KUKA KRL program: repair_test.src, repair_test.dat

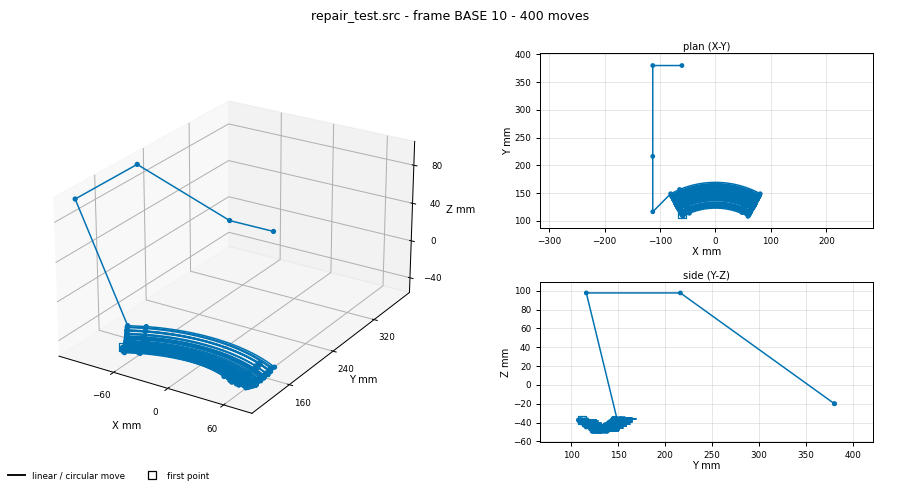
[picture p0: tool path of repair_test.src in frame BASE 10, 400 of 403 moves have a stored position in this frame; points joined in program order, loops and branches not executed]
--- repair_test.src ---
&ACCESS RVP1
&REL 1217
&PARAM WOPTRAJECTORYID = 2
&PARAM WOPTEMPLATENAME = WopCoreTemplatePath
&PARAM DISKPATH = KRC:\R1\Program\Working Paths
DEF  repair_test ( )

;FOLD INI
InitWopCoreSrc(#Init_Trajectory)
;ENDFOLD (INI)

;FOLD Manual mode
IF X_Rob_InManu THEN
;Write here the code executed only in manual mode

ENDIF
;ENDFOLD

X_Prod_En_Cours[2]=TRUE

;FOLD PTP PT_LoopPos1 Vel=10 % DEFAULT Tool[1]:Gun Base[0];%{PE}
;FOLD Parameters ;%{h}
;Params IlfProvider=kukaroboter.basistech.inlineforms.movement.old; Kuka.IsGlobalPoint=False; Kuka.PointName=PT_LoopPos1; Kuka.BlendingEnabled=False; Kuka.MoveDataPtpName=DEFAULT; Kuka.VelocityPtp=10; Kuka.CurrentCDSetIndex=0; Kuka.MovementParameterFieldEnabled=True; IlfCommand=PTP
;ENDFOLD
$BWDSTART = FALSE
PDAT_ACT = PDEFAULT
FDAT_ACT = FPT_LoopPos1
BAS(#PTP_PARAMS, 10.0)
SET_CD_PARAMS (0)
PTP XPT_LoopPos1
;ENDFOLD



;FOLD CHECK DAT-FILE GENERATION NUMBER
  IF APP_GENNUMBER <> 215375 THEN
    LOOP
      MsgQuit("InconsistenceSRCandDAT",,,,1)
      HALT
    ENDLOOP
  ENDIF
;ENDFOLD

;fold Jobinfo
;Job information: repair_test
;Product : 3.1.0.28784
;Date: 2026-09-17-14_00
;Project name: repair_test
;Author: Alhadi Zidan
;Company: CRITT-TJFU
;Division: CSAMProj
;Comment: Autogenerated CSAM Path
;endfold

; --- GLOBAL BLENDING OVERRIDES ---
$APO.CDIS = 1.0  ; Distance blending radius (mm)
$APO.CVEL = 100  ; Velocity blending (%)
$APO.CORI = 5.0  ; Orientation blending (degrees)
$ADVANCE = 5
;FOLD PTP P0 Vel=100 % P0 Tool[2] Base[10] ;%{PE}
;FOLD Parameters ;%{h}
;Params IlfProvider=kukaroboter.basistech.inlineforms.movement.old; Kuka.IsGlobalPoint=False; Kuka.PointName=P0; Kuka.BlendingEnabled=FALSE; Kuka.MoveDataName=PDATP0; Kuka.VelocityPath=100; Kuka.CurrentCDSetIndex=0; Kuka.MovementParameterFieldEnabled=True; IlfCommand=PTP
;ENDFOLD
$BWDSTART = FALSE
PDAT_ACT=PPDATP0
FDAT_ACT=FP0
BAS (#PTP_PARAMS,100)
SET_CD_PARAMS (0)
PTP XP0

;ENDFOLD
Routine_0()
;FOLD PTP PT_LoopPos1 Vel=60 % DEFAULT Tool[1]:Gun Base[0];%{{PE}}
;FOLD Parameters ;%{{h}}
;Params IlfProvider=kukaroboter.basistech.inlineforms.movement.old; Kuka.IsGlobalPoint=False; Kuka.PointName=PT_LoopPos1; Kuka.BlendingEnabled=False; Kuka.MoveDataPtpName=DEFAULT; Kuka.VelocityPtp=10; Kuka.CurrentCDSetIndex=0; Kuka.MovementParameterFieldEnabled=True; IlfCommand=PTP
;ENDFOLD
$BWDSTART = FALSE
PDAT_ACT = PDEFAULT
FDAT_ACT = FPT_LoopPos1
BAS(#PTP_PARAMS, 60.0)
SET_CD_PARAMS (0)
PTP XPT_LoopPos1
;ENDFOLD
END

; --- Routine for substrate 0 ---
DEF Routine_0()
;FOLD LIN P1 CONT Vel=1 m/s CPDATP1 Tool[2] Base[10] ;%{PE}
;FOLD Parameters ;%{h}
;Params IlfProvider=kukaroboter.basistech.inlineforms.movement.old; Kuka.IsGlobalPoint=False; Kuka.PointName=P1; Kuka.BlendingEnabled=TRUE; Kuka.MoveDataName=CPDATP1; Kuka.VelocityPath=1; Kuka.CurrentCDSetIndex=0; Kuka.MovementParameterFieldEnabled=True; IlfCommand=LIN
;ENDFOLD
$BWDSTART = FALSE
LDAT_ACT=LCPDATP1
FDAT_ACT=FP1
BAS (#CP_PARAMS,1)
SET_CD_PARAMS (0)
LIN XP1 C_DIS

;ENDFOLD
;FOLD CIRC CAux2 CDes2 CONT Vel=0.1 m/s CPDATC2 Tool[2] Base[10] ;%{PE}
;FOLD Parameters ;%{h}
;Params IlfProvider=kukaroboter.basistech.inlineforms.movement.old; Kuka.IsGlobalPoint=False; Kuka.PointName=CDes2; Kuka.BlendingEnabled=TRUE; Kuka.MoveDataName=CPDATC2; Kuka.VelocityPath=0.1; Kuka.CurrentCDSetIndex=0; Kuka.MovementParameterFieldEnabled=True; IlfCommand=LIN
;ENDFOLD
$BWDSTART = FALSE
LDAT_ACT=LCPDATC2
FDAT_ACT=FC2
$ORI_TYPE = #VAR
$CIRC_TYPE = #PATH
BAS (#CP_PARAMS,0.1)
SET_CD_PARAMS (0)
CIRC XCAux2, XCDes2 C_DIS

;ENDFOLD
;FOLD LIN P3 CONT Vel=1 m/s CPDATP3 Tool[2] Base[10] ;%{PE}
;FOLD Parameters ;%{h}
;Params IlfProvider=kukaroboter.basistech.inlineforms.movement.old; Kuka.IsGlobalPoint=False; Kuka.PointName=P3; Kuka.BlendingEnabled=TRUE; Kuka.MoveDataName=CPDATP3; Kuka.VelocityPath=1; Kuka.CurrentCDSetIndex=0; Kuka.MovementParameterFieldEnabled=True; IlfCommand=LIN
;ENDFOLD
$BWDSTART = FALSE
LDAT_ACT=LCPDATP3
FDAT_ACT=FP3
BAS (#CP_PARAMS,1)
SET_CD_PARAMS (0)
LIN XP3 C_DIS

;ENDFOLD
;FOLD LIN P4 CONT Vel=1 m/s CPDATP4 Tool[2] Base[10] ;%{PE}
;FOLD Parameters ;%{h}
;Params IlfProvider=kukaroboter.basistech.inlineforms.movement.old; Kuka.IsGlobalPoint=False; Kuka.PointName=P4; Kuka.BlendingEnabled=TRUE; Kuka.MoveDataName=CPDATP4; Kuka.VelocityPath=1; Kuka.CurrentCDSetIndex=0; Kuka.MovementParameterFieldEnabled=True; IlfCommand=LIN
;ENDFOLD
$BWDSTART = FALSE
LDAT_ACT=LCPDATP4
FDAT_ACT=FP4
BAS (#CP_PARAMS,1)
SET_CD_PARAMS (0)
LIN XP4 C_DIS

;ENDFOLD
;FOLD CIRC CAux5 CDes5 CONT Vel=0.1 m/s CPDATC5 Tool[2] Base[10] ;%{PE}
;FOLD Parameters ;%{h}
;Params IlfProvider=kukaroboter.basistech.inlineforms.movement.old; Kuka.IsGlobalPoint=False; Kuka.PointName=CDes5; Kuka.BlendingEnabled=TRUE; Kuka.MoveDataName=CPDATC5; Kuka.VelocityPath=0.1; Kuka.CurrentCDSetIndex=0; Kuka.MovementParameterFieldEnabled=True; IlfCommand=LIN
;ENDFOLD
$BWDSTART = FALSE
LDAT_ACT=LCPDATC5
FDAT_ACT=FC5
$ORI_TYPE = #VAR
$CIRC_TYPE = #PATH
BAS (#CP_PARAMS,0.1)
SET_CD_PARAMS (0)
CIRC XCAux5, XCDes5 C_DIS

;ENDFOLD
;FOLD LIN P6 CONT Vel=1 m/s CPDATP6 Tool[2] Base[10] ;%{PE}
;FOLD Parameters ;%{h}
;Params IlfProvider=kukaroboter.basistech.inlineforms.movement.old; Kuka.IsGlobalPoint=False; Kuka.PointName=P6; Kuka.BlendingEnabled=TRUE; Kuka.MoveDataName=CPDATP6; Kuka.VelocityPath=1; Kuka.CurrentCDSetIndex=0; Kuka.MovementParameterFieldEnabled=True; IlfCommand=LIN
;ENDFOLD
$BWDSTART = FALSE
LDAT_ACT=LCPDATP6
FDAT_ACT=FP6
BAS (#CP_PARAMS,1)
SET_CD_PARAMS (0)
LIN XP6 C_DIS

;ENDFOLD
;FOLD LIN P7 CONT Vel=1 m/s CPDATP7 Tool[2] Base[10] ;%{PE}
;FOLD Parameters ;%{h}
;Params IlfProvider=kukaroboter.basistech.inlineforms.movement.old; Kuka.IsGlobalPoint=False; Kuka.PointName=P7; Kuka.BlendingEnabled=TRUE; Kuka.MoveDataName=CPDATP7; Kuka.VelocityPath=1; Kuka.CurrentCDSetIndex=0; Kuka.MovementParameterFieldEnabled=True; IlfCommand=LIN
;ENDFOLD
$BWDSTART = FALSE
LDAT_ACT=LCPDATP7
FDAT_ACT=FP7
BAS (#CP_PARAMS,1)
SET_CD_PARAMS (0)
LIN XP7 C_DIS

;ENDFOLD
;FOLD CIRC CAux8 CDes8 CONT Vel=0.1 m/s CPDATC8 Tool[2] Base[10] ;%{PE}
;FOLD Parameters ;%{h}
;Params IlfProvider=kukaroboter.basistech.inlineforms.movement.old; Kuka.IsGlobalPoint=False; Kuka.PointName=CDes8; Kuka.BlendingEnabled=TRUE; Kuka.MoveDataName=CPDATC8; Kuka.VelocityPath=0.1; Kuka.CurrentCDSetIndex=0; Kuka.MovementParameterFieldEnabled=True; IlfCommand=LIN
;ENDFOLD
$BWDSTART = FALSE
LDAT_ACT=LCPDATC8
FDAT_ACT=FC8
$ORI_TYPE = #VAR
$CIRC_TYPE = #PATH
BAS (#CP_PARAMS,0.1)
SET_CD_PARAMS (0)
CIRC XCAux8, XCDes8 C_DIS

;ENDFOLD
;FOLD LIN P9 CONT Vel=1 m/s CPDATP9 Tool[2] Base[10] ;%{PE}
;FOLD Parameters ;%{h}
;Params IlfProvider=kukaroboter.basistech.inlineforms.movement.old; Kuka.IsGlobalPoint=False; Kuka.PointName=P9; Kuka.BlendingEnabled=TRUE; Kuka.MoveDataName=CPDATP9; Kuka.VelocityPath=1; Kuka.CurrentCDSetIndex=0; Kuka.MovementParameterFieldEnabled=True; IlfCommand=LIN
;ENDFOLD
$BWDSTART = FALSE
LDAT_ACT=LCPDATP9
FDAT_ACT=FP9
BAS (#CP_PARAMS,1)
SET_CD_PARAMS (0)
LIN XP9 C_DIS

;ENDFOLD
;FOLD LIN P10 CONT Vel=1 m/s CPDATP10 Tool[2] Base[10] ;%{PE}
;FOLD Parameters ;%{h}
;Params IlfProvider=kukaroboter.basistech.inlineforms.movement.old; Kuka.IsGlobalPoint=False; Kuka.PointName=P10; Kuka.BlendingEnabled=TRUE; Kuka.MoveDataName=CPDATP10; Kuka.VelocityPath=1; Kuka.CurrentCDSetIndex=0; Kuka.MovementParameterFieldEnabled=True; IlfCommand=LIN
;ENDFOLD
$BWDSTART = FALSE
LDAT_ACT=LCPDATP10
FDAT_ACT=FP10
BAS (#CP_PARAMS,1)
SET_CD_PARAMS (0)
LIN XP10 C_DIS

;ENDFOLD
;FOLD CIRC CAux11 CDes11 CONT Vel=0.1 m/s CPDATC11 Tool[2] Base[10] ;%{PE}
;FOLD Parameters ;%{h}
;Params IlfProvider=kukaroboter.basistech.inlineforms.movement.old; Kuka.IsGlobalPoint=False; Kuka.PointName=CDes11; Kuka.BlendingEnabled=TRUE; Kuka.MoveDataName=CPDATC11; Kuka.VelocityPath=0.1; Kuka.CurrentCDSetIndex=0; Kuka.MovementParameterFieldEnabled=True; IlfCommand=LIN
;ENDFOLD
$BWDSTART = FALSE
LDAT_ACT=LCPDATC11
FDAT_ACT=FC11
$ORI_TYPE = #VAR
$CIRC_TYPE = #PATH
BAS (#CP_PARAMS,0.1)
SET_CD_PARAMS (0)
CIRC XCAux11, XCDes11 C_DIS

;ENDFOLD
;FOLD LIN P12 CONT Vel=1 m/s CPDATP12 Tool[2] Base[10] ;%{PE}
;FOLD Parameters ;%{h}
;Params IlfProvider=kukaroboter.basistech.inlineforms.movement.old; Kuka.IsGlobalPoint=False; Kuka.PointName=P12; Kuka.BlendingEnabled=TRUE; Kuka.MoveDataName=CPDATP12; Kuka.VelocityPath=1; Kuka.CurrentCDSetIndex=0; Kuka.MovementParameterFieldEnabled=True; IlfCommand=LIN
;ENDFOLD
$BWDSTART = FALSE
LDAT_ACT=LCPDATP12
FDAT_ACT=FP12
BAS (#CP_PARAMS,1)
SET_CD_PARAMS (0)
LIN XP12 C_DIS

;ENDFOLD
;FOLD LIN P13 CONT Vel=1 m/s CPDATP13 Tool[2] Base[10] ;%{PE}
;FOLD Parameters ;%{h}
;Params IlfProvider=kukaroboter.basistech.inlineforms.movement.old; Kuka.IsGlobalPoint=False; Kuka.PointName=P13; Kuka.BlendingEnabled=TRUE; Kuka.MoveDataName=CPDATP13; Kuka.VelocityPath=1; Kuka.CurrentCDSetIndex=0; Kuka.MovementParameterFieldEnabled=True; IlfCommand=LIN
;ENDFOLD
$BWDSTART = FALSE
LDAT_ACT=LCPDATP13
FDAT_ACT=FP13
BAS (#CP_PARAMS,1)
SET_CD_PARAMS (0)
LIN XP13 C_DIS

;ENDFOLD
;FOLD CIRC CAux14 CDes14 CONT Vel=0.1 m/s CPDATC14 Tool[2] Base[10] ;%{PE}
;FOLD Parameters ;%{h}
;Params IlfProvider=kukaroboter.basistech.inlineforms.movement.old; Kuka.IsGlobalPoint=False; Kuka.PointName=CDes14; Kuka.BlendingEnabled=TRUE; Kuka.MoveDataName=CPDATC14; Kuka.VelocityPath=0.1; Kuka.CurrentCDSetIndex=0; Kuka.MovementParameterFieldEnabled=True; IlfCommand=LIN
;ENDFOLD
$BWDSTART = FALSE
LDAT_ACT=LCPDATC14
FDAT_ACT=FC14
$ORI_TYPE = #VAR
$CIRC_TYPE = #PATH
BAS (#CP_PARAMS,0.1)
SET_CD_PARAMS (0)
CIRC XCAux14, XCDes14 C_DIS

;ENDFOLD
;FOLD LIN P15 CONT Vel=1 m/s CPDATP15 Tool[2] Base[10] ;%{PE}
;FOLD Parameters ;%{h}
;Params IlfProvider=kukaroboter.basistech.inlineforms.movement.old; Kuka.IsGlobalPoint=False; Kuka.PointName=P15; Kuka.BlendingEnabled=TRUE; Kuka.MoveDataName=CPDATP15; Kuka.VelocityPath=1; Kuka.CurrentCDSetIndex=0; Kuka.MovementParameterFieldEnabled=True; IlfCommand=LIN
;ENDFOLD
$BWDSTART = FALSE
LDAT_ACT=LCPDATP15
FDAT_ACT=FP15
BAS (#CP_PARAMS,1)
SET_CD_PARAMS (0)
LIN XP15 C_DIS

;ENDFOLD
;FOLD LIN P16 CONT Vel=1 m/s CPDATP16 Tool[2] Base[10] ;%{PE}
;FOLD Parameters ;%{h}
;Params IlfProvider=kukaroboter.basistech.inlineforms.movement.old; Kuka.IsGlobalPoint=False; Kuka.PointName=P16; Kuka.BlendingEnabled=TRUE; Kuka.MoveDataName=CPDATP16; Kuka.VelocityPath=1; Kuka.CurrentCDSetIndex=0; Kuka.MovementParameterFieldEnabled=True; IlfCommand=LIN
;ENDFOLD
$BWDSTART = FALSE
LDAT_ACT=LCPDATP16
FDAT_ACT=FP16
BAS (#CP_PARAMS,1)
SET_CD_PARAMS (0)
LIN XP16 C_DIS

;ENDFOLD
;FOLD CIRC CAux17 CDes17 CONT Vel=0.1 m/s CPDATC17 Tool[2] Base[10] ;%{PE}
;FOLD Parameters ;%{h}
;Params IlfProvider=kukaroboter.basistech.inlineforms.movement.old; Kuka.IsGlobalPoint=False; Kuka.PointName=CDes17; Kuka.BlendingEnabled=TRUE; Kuka.MoveDataName=CPDATC17; Kuka.VelocityPath=0.1; Kuka.CurrentCDSetIndex=0; Kuka.MovementParameterFieldEnabled=True; IlfCommand=LIN
;ENDFOLD
$BWDSTART = FALSE
LDAT_ACT=LCPDATC17
FDAT_ACT=FC17
$ORI_TYPE = #VAR
$CIRC_TYPE = #PATH
BAS (#CP_PARAMS,0.1)
SET_CD_PARAMS (0)
CIRC XCAux17, XCDes17 C_DIS

;ENDFOLD
;FOLD LIN P18 CONT Vel=1 m/s CPDATP18 Tool[2] Base[10] ;%{PE}
;FOLD Parameters ;%{h}
;Params IlfProvider=kukaroboter.basistech.inlineforms.movement.old; Kuka.IsGlobalPoint=False; Kuka.PointName=P18; Kuka.BlendingEnabled=TRUE; Kuka.MoveDataName=CPDATP18; Kuka.VelocityPath=1; Kuka.CurrentCDSetIndex=0; Kuka.MovementParameterFieldEnabled=True; IlfCommand=LIN
;ENDFOLD
$BWDSTART = FALSE
LDAT_ACT=LCPDATP18
FDAT_ACT=FP18
BAS (#CP_PARAMS,1)
SET_CD_PARAMS (0)
LIN XP18 C_DIS

;ENDFOLD
;FOLD LIN P19 CONT Vel=1 m/s CPDATP19 Tool[2] Base[10] ;%{PE}
;FOLD Parameters ;%{h}
;Params IlfProvider=kukaroboter.basistech.inlineforms.movement.old; Kuka.IsGlobalPoint=False; Kuka.PointName=P19; Kuka.BlendingEnabled=TRUE; Kuka.MoveDataName=CPDATP19; Kuka.VelocityPath=1; Kuka.CurrentCDSetIndex=0; Kuka.MovementParameterFieldEnabled=True; IlfCommand=LIN
;ENDFOLD
$BWDSTART = FALSE
LDAT_ACT=LCPDATP19
FDAT_ACT=FP19
BAS (#CP_PARAMS,1)
SET_CD_PARAMS (0)
LIN XP19 C_DIS

;ENDFOLD
;FOLD CIRC CAux20 CDes20 CONT Vel=0.1 m/s CPDATC20 Tool[2] Base[10] ;%{PE}
;FOLD Parameters ;%{h}
;Params IlfProvider=kukaroboter.basistech.inlineforms.movement.old; Kuka.IsGlobalPoint=False; Kuka.PointName=CDes20; Kuka.BlendingEnabled=TRUE; Kuka.MoveDataName=CPDATC20; Kuka.VelocityPath=0.1; Kuka.CurrentCDSetIndex=0; Kuka.MovementParameterFieldEnabled=True; IlfCommand=LIN
;ENDFOLD
$BWDSTART = FALSE
LDAT_ACT=LCPDATC20
FDAT_ACT=FC20
$ORI_TYPE = #VAR
$CIRC_TYPE = #PATH
BAS (#CP_PARAMS,0.1)
SET_CD_PARAMS (0)
CIRC XCAux20, XCDes20 C_DIS

;ENDFOLD
;FOLD LIN P21 CONT Vel=1 m/s CPDATP21 Tool[2] Base[10] ;%{PE}
;FOLD Parameters ;%{h}
;Params IlfProvider=kukaroboter.basistech.inlineforms.movement.old; Kuka.IsGlobalPoint=False; Kuka.PointName=P21; Kuka.BlendingEnabled=TRUE; Kuka.MoveDataName=CPDATP21; Kuka.VelocityPath=1; Kuka.CurrentCDSetIndex=0; Kuka.MovementParameterFieldEnabled=True; IlfCommand=LIN
;ENDFOLD
$BWDSTART = FALSE
LDAT_ACT=LCPDATP21
FDAT_ACT=FP21
BAS (#CP_PARAMS,1)
SET_CD_PARAMS (0)
LIN XP21 C_DIS

;ENDFOLD
;FOLD LIN P22 CONT Vel=1 m/s CPDATP22 Tool[2] Base[10] ;%{PE}
;FOLD Parameters ;%{h}
;Params IlfProvider=kukaroboter.basistech.inlineforms.movement.old; Kuka.IsGlobalPoint=False; Kuka.PointName=P22; Kuka.BlendingEnabled=TRUE; Kuka.MoveDataName=CPDATP22; Kuka.VelocityPath=1; Kuka.CurrentCDSetIndex=0; Kuka.MovementParameterFieldEnabled=True; IlfCommand=LIN
;ENDFOLD
$BWDSTART = FALSE
LDAT_ACT=LCPDATP22
FDAT_ACT=FP22
BAS (#CP_PARAMS,1)
SET_CD_PARAMS (0)
LIN XP22 C_DIS

;ENDFOLD
;FOLD CIRC CAux23 CDes23 CONT Vel=0.1 m/s CPDATC23 Tool[2] Base[10] ;%{PE}
;FOLD Parameters ;%{h}
;Params IlfProvider=kukaroboter.basistech.inlineforms.movement.old; Kuka.IsGlobalPoint=False; Kuka.PointName=CDes23; Kuka.BlendingEnabled=TRUE; Kuka.MoveDataName=CPDATC23; Kuka.VelocityPath=0.1; Kuka.CurrentCDSetIndex=0; Kuka.MovementParameterFieldEnabled=True; IlfCommand=LIN
;ENDFOLD
$BWDSTART = FALSE
LDAT_ACT=LCPDATC23
FDAT_ACT=FC23
$ORI_TYPE = #VAR
$CIRC_TYPE = #PATH
BAS (#CP_PARAMS,0.1)
SET_CD_PARAMS (0)
CIRC XCAux23, XCDes23 C_DIS

;ENDFOLD
;FOLD LIN P24 CONT Vel=1 m/s CPDATP24 Tool[2] Base[10] ;%{PE}
;FOLD Parameters ;%{h}
;Params IlfProvider=kukaroboter.basistech.inlineforms.movement.old; Kuka.IsGlobalPoint=False; Kuka.PointName=P24; Kuka.BlendingEnabled=TRUE; Kuka.MoveDataName=CPDATP24; Kuka.VelocityPath=1; Kuka.CurrentCDSetIndex=0; Kuka.MovementParameterFieldEnabled=True; IlfCommand=LIN
;ENDFOLD
$BWDSTART = FALSE
LDAT_ACT=LCPDATP24
FDAT_ACT=FP24
BAS (#CP_PARAMS,1)
SET_CD_PARAMS (0)
LIN XP24 C_DIS

;ENDFOLD
;FOLD LIN P25 CONT Vel=1 m/s CPDATP25 Tool[2] Base[10] ;%{PE}
;FOLD Parameters ;%{h}
;Params IlfProvider=kukaroboter.basistech.inlineforms.movement.old; Kuka.IsGlobalPoint=False; Kuka.PointName=P25; Kuka.BlendingEnabled=TRUE; Kuka.MoveDataName=CPDATP25; Kuka.VelocityPath=1; Kuka.CurrentCDSetIndex=0; Kuka.MovementParameterFieldEnabled=True; IlfCommand=LIN
;ENDFOLD
$BWDSTART = FALSE
LDAT_ACT=LCPDATP25
FDAT_ACT=FP25
BAS (#CP_PARAMS,1)
SET_CD_PARAMS (0)
LIN XP25 C_DIS

;ENDFOLD
;FOLD CIRC CAux26 CDes26 CONT Vel=0.1 m/s CPDATC26 Tool[2] Base[10] ;%{PE}
;FOLD Parameters ;%{h}
;Params IlfProvider=kukaroboter.basistech.inlineforms.movement.old; Kuka.IsGlobalPoint=False; Kuka.PointName=CDes26; Kuka.BlendingEnabled=TRUE; Kuka.MoveDataName=CPDATC26; Kuka.VelocityPath=0.1; Kuka.CurrentCDSetIndex=0; Kuka.MovementParameterFieldEnabled=True; IlfCommand=LIN
;ENDFOLD
$BWDSTART = FALSE
LDAT_ACT=LCPDATC26
FDAT_ACT=FC26
$ORI_TYPE = #VAR
$CIRC_TYPE = #PATH
BAS (#CP_PARAMS,0.1)
SET_CD_PARAMS (0)
CIRC XCAux26, XCDes26 C_DIS

;ENDFOLD
;FOLD LIN P27 CONT Vel=1 m/s CPDATP27 Tool[2] Base[10] ;%{PE}
;FOLD Parameters ;%{h}
;Params IlfProvider=kukaroboter.basistech.inlineforms.movement.old; Kuka.IsGlobalPoint=False; Kuka.PointName=P27; Kuka.BlendingEnabled=TRUE; Kuka.MoveDataName=CPDATP27; Kuka.VelocityPath=1; Kuka.CurrentCDSetIndex=0; Kuka.MovementParameterFieldEnabled=True; IlfCommand=LIN
;ENDFOLD
$BWDSTART = FALSE
LDAT_ACT=LCPDATP27
FDAT_ACT=FP27
BAS (#CP_PARAMS,1)
SET_CD_PARAMS (0)
LIN XP27 C_DIS

;ENDFOLD
;FOLD LIN P28 CONT Vel=1 m/s CPDATP28 Tool[2] Base[10] ;%{PE}
;FOLD Parameters ;%{h}
;Params IlfProvider=kukaroboter.basistech.inlineforms.movement.old; Kuka.IsGlobalPoint=False; Kuka.PointName=P28; Kuka.BlendingEnabled=TRUE; Kuka.MoveDataName=CPDATP28; Kuka.VelocityPath=1; Kuka.CurrentCDSetIndex=0; Kuka.MovementParameterFieldEnabled=True; IlfCommand=LIN
;ENDFOLD
$BWDSTART = FALSE
LDAT_ACT=LCPDATP28
FDAT_ACT=FP28
BAS (#CP_PARAMS,1)
SET_CD_PARAMS (0)
LIN XP28 C_DIS

;ENDFOLD
;FOLD CIRC CAux29 CDes29 CONT Vel=0.1 m/s CPDATC29 Tool[2] Base[10] ;%{PE}
;FOLD Parameters ;%{h}
;Params IlfProvider=kukaroboter.basistech.inlineforms.movement.old; Kuka.IsGlobalPoint=False; Kuka.PointName=CDes29; Kuka.BlendingEnabled=TRUE; Kuka.MoveDataName=CPDATC29; Kuka.VelocityPath=0.1; Kuka.CurrentCDSetIndex=0; Kuka.MovementParameterFieldEnabled=True; IlfCommand=LIN
;ENDFOLD
$BWDSTART = FALSE
LDAT_ACT=LCPDATC29
FDAT_ACT=FC29
$ORI_TYPE = #VAR
$CIRC_TYPE = #PATH
BAS (#CP_PARAMS,0.1)
SET_CD_PARAMS (0)
CIRC XCAux29, XCDes29 C_DIS

;ENDFOLD
;FOLD LIN P30 CONT Vel=1 m/s CPDATP30 Tool[2] Base[10] ;%{PE}
;FOLD Parameters ;%{h}
;Params IlfProvider=kukaroboter.basistech.inlineforms.movement.old; Kuka.IsGlobalPoint=False; Kuka.PointName=P30; Kuka.BlendingEnabled=TRUE; Kuka.MoveDataName=CPDATP30; Kuka.VelocityPath=1; Kuka.CurrentCDSetIndex=0; Kuka.MovementParameterFieldEnabled=True; IlfCommand=LIN
;ENDFOLD
$BWDSTART = FALSE
LDAT_ACT=LCPDATP30
FDAT_ACT=FP30
BAS (#CP_PARAMS,1)
SET_CD_PARAMS (0)
LIN XP30 C_DIS

;ENDFOLD
;FOLD LIN P31 CONT Vel=1 m/s CPDATP31 Tool[2] Base[10] ;%{PE}
;FOLD Parameters ;%{h}
;Params IlfProvider=kukaroboter.basistech.inlineforms.movement.old; Kuka.IsGlobalPoint=False; Kuka.PointName=P31; Kuka.BlendingEnabled=TRUE; Kuka.MoveDataName=CPDATP31; Kuka.VelocityPath=1; Kuka.CurrentCDSetIndex=0; Kuka.MovementParameterFieldEnabled=True; IlfCommand=LIN
;ENDFOLD
$BWDSTART = FALSE
LDAT_ACT=LCPDATP31
FDAT_ACT=FP31
BAS (#CP_PARAMS,1)
SET_CD_PARAMS (0)
LIN XP31 C_DIS

;ENDFOLD
;FOLD CIRC CAux32 CDes32 CONT Vel=0.1 m/s CPDATC32 Tool[2] Base[10] ;%{PE}
;FOLD Parameters ;%{h}
;Params IlfProvider=kukaroboter.basistech.inlineforms.movement.old; Kuka.IsGlobalPoint=False; Kuka.PointName=CDes32; Kuka.BlendingEnabled=TRUE; Kuka.MoveDataName=CPDATC32; Kuka.VelocityPath=0.1; Kuka.CurrentCDSetIndex=0; Kuka.MovementParameterFieldEnabled=True; IlfCommand=LIN
;ENDFOLD
$BWDSTART = FALSE
LDAT_ACT=LCPDATC32
FDAT_ACT=FC32
$ORI_TYPE = #VAR
$CIRC_TYPE = #PATH
BAS (#CP_PARAMS,0.1)
SET_CD_PARAMS (0)
CIRC XCAux32, XCDes32 C_DIS

;ENDFOLD
;FOLD LIN P33 CONT Vel=1 m/s CPDATP33 Tool[2] Base[10] ;%{PE}
;FOLD Parameters ;%{h}
;Params IlfProvider=kukaroboter.basistech.inlineforms.movement.old; Kuka.IsGlobalPoint=False; Kuka.PointName=P33; Kuka.BlendingEnabled=TRUE; Kuka.MoveDataName=CPDATP33; Kuka.VelocityPath=1; Kuka.CurrentCDSetIndex=0; Kuka.MovementParameterFieldEnabled=True; IlfCommand=LIN
;ENDFOLD
$BWDSTART = FALSE
LDAT_ACT=LCPDATP33
FDAT_ACT=FP33
BAS (#CP_PARAMS,1)
SET_CD_PARAMS (0)
LIN XP33 C_DIS

;ENDFOLD
;FOLD LIN P34 CONT Vel=1 m/s CPDATP34 Tool[2] Base[10] ;%{PE}
;FOLD Parameters ;%{h}
;Params IlfProvider=kukaroboter.basistech.inlineforms.movement.old; Kuka.IsGlobalPoint=False; Kuka.PointName=P34; Kuka.BlendingEnabled=TRUE; Kuka.MoveDataName=CPDATP34; Kuka.VelocityPath=1; Kuka.CurrentCDSetIndex=0; Kuka.MovementParameterFieldEnabled=True; IlfCommand=LIN
;ENDFOLD
$BWDSTART = FALSE
LDAT_ACT=LCPDATP34
FDAT_ACT=FP34
BAS (#CP_PARAMS,1)
SET_CD_PARAMS (0)
LIN XP34 C_DIS

;ENDFOLD
;FOLD CIRC CAux35 CDes35 CONT Vel=0.1 m/s CPDATC35 Tool[2] Base[10] ;%{PE}
;FOLD Parameters ;%{h}
;Params IlfProvider=kukaroboter.basistech.inlineforms.movement.old; Kuka.IsGlobalPoint=False; Kuka.PointName=CDes35; Kuka.BlendingEnabled=TRUE; Kuka.MoveDataName=CPDATC35; Kuka.VelocityPath=0.1; Kuka.CurrentCDSetIndex=0; Kuka.MovementParameterFieldEnabled=True; IlfCommand=LIN
;ENDFOLD
$BWDSTART = FALSE
LDAT_ACT=LCPDATC35
FDAT_ACT=FC35
$ORI_TYPE = #VAR
$CIRC_TYPE = #PATH
BAS (#CP_PARAMS,0.1)
SET_CD_PARAMS (0)
CIRC XCAux35, XCDes35 C_DIS

;ENDFOLD
;FOLD LIN P36 CONT Vel=1 m/s CPDATP36 Tool[2] Base[10] ;%{PE}
;FOLD Parameters ;%{h}
;Params IlfProvider=kukaroboter.basistech.inlineforms.movement.old; Kuka.IsGlobalPoint=False; Kuka.PointName=P36; Kuka.BlendingEnabled=TRUE; Kuka.MoveDataName=CPDATP36; Kuka.VelocityPath=1; Kuka.CurrentCDSetIndex=0; Kuka.MovementParameterFieldEnabled=True; IlfCommand=LIN
;ENDFOLD
$BWDSTART = FALSE
LDAT_ACT=LCPDATP36
FDAT_ACT=FP36
BAS (#CP_PARAMS,1)
SET_CD_PARAMS (0)
LIN XP36 C_DIS

;ENDFOLD
;FOLD LIN P37 CONT Vel=1 m/s CPDATP37 Tool[2] Base[10] ;%{PE}
;FOLD Parameters ;%{h}
;Params IlfProvider=kukaroboter.basistech.inlineforms.movement.old; Kuka.IsGlobalPoint=False; Kuka.PointName=P37; Kuka.BlendingEnabled=TRUE; Kuka.MoveDataName=CPDATP37; Kuka.VelocityPath=1; Kuka.CurrentCDSetIndex=0; Kuka.MovementParameterFieldEnabled=True; IlfCommand=LIN
;ENDFOLD
$BWDSTART = FALSE
LDAT_ACT=LCPDATP37
FDAT_ACT=FP37
BAS (#CP_PARAMS,1)
SET_CD_PARAMS (0)
LIN XP37 C_DIS

;ENDFOLD
;FOLD CIRC CAux38 CDes38 CONT Vel=0.1 m/s CPDATC38 Tool[2] Base[10] ;%{PE}
;FOLD Parameters ;%{h}
;Params IlfProvider=kukaroboter.basistech.inlineforms.movement.old; Kuka.IsGlobalPoint=False; Kuka.PointName=CDes38; Kuka.BlendingEnabled=TRUE; Kuka.MoveDataName=CPDATC38; Kuka.VelocityPath=0.1; Kuka.CurrentCDSetIndex=0; Kuka.MovementParameterFieldEnabled=True; IlfCommand=LIN
;ENDFOLD
$BWDSTART = FALSE
LDAT_ACT=LCPDATC38
FDAT_ACT=FC38
$ORI_TYPE = #VAR
$CIRC_TYPE = #PATH
BAS (#CP_PARAMS,0.1)
SET_CD_PARAMS (0)
CIRC XCAux38, XCDes38 C_DIS

;ENDFOLD
;FOLD LIN P39 CONT Vel=1 m/s CPDATP39 Tool[2] Base[10] ;%{PE}
;FOLD Parameters ;%{h}
;Params IlfProvider=kukaroboter.basistech.inlineforms.movement.old; Kuka.IsGlobalPoint=False; Kuka.PointName=P39; Kuka.BlendingEnabled=TRUE; Kuka.MoveDataName=CPDATP39; Kuka.VelocityPath=1; Kuka.CurrentCDSetIndex=0; Kuka.MovementParameterFieldEnabled=True; IlfCommand=LIN
;ENDFOLD
$BWDSTART = FALSE
LDAT_ACT=LCPDATP39
FDAT_ACT=FP39
BAS (#CP_PARAMS,1)
SET_CD_PARAMS (0)
LIN XP39 C_DIS

;ENDFOLD
;FOLD LIN P40 CONT Vel=1 m/s CPDATP40 Tool[2] Base[10] ;%{PE}
;FOLD Parameters ;%{h}
;Params IlfProvider=kukaroboter.basistech.inlineforms.movement.old; Kuka.IsGlobalPoint=False; Kuka.PointName=P40; Kuka.BlendingEnabled=TRUE; Kuka.MoveDataName=CPDATP40; Kuka.VelocityPath=1; Kuka.CurrentCDSetIndex=0; Kuka.MovementParameterFieldEnabled=True; IlfCommand=LIN
;ENDFOLD
$BWDSTART = FALSE
LDAT_ACT=LCPDATP40
FDAT_ACT=FP40
BAS (#CP_PARAMS,1)
SET_CD_PARAMS (0)
LIN XP40 C_DIS

;ENDFOLD
;FOLD CIRC CAux41 CDes41 CONT Vel=0.1 m/s CPDATC41 Tool[2] Base[10] ;%{PE}
;FOLD Parameters ;%{h}
;Params IlfProvider=kukaroboter.basistech.inlineforms.movement.old; Kuka.IsGlobalPoint=False; Kuka.PointName=CDes41; Kuka.BlendingEnabled=TRUE; Kuka.MoveDataName=CPDATC41; Kuka.VelocityPath=0.1; Kuka.CurrentCDSetIndex=0; Kuka.MovementParameterFieldEnabled=True; IlfCommand=LIN
;ENDFOLD
$BWDSTART = FALSE
LDAT_ACT=LCPDATC41
FDAT_ACT=FC41
$ORI_TYPE = #VAR
$CIRC_TYPE = #PATH
BAS (#CP_PARAMS,0.1)
SET_CD_PARAMS (0)
CIRC XCAux41, XCDes41 C_DIS

;ENDFOLD
;FOLD LIN P42 CONT Vel=1 m/s CPDATP42 Tool[2] Base[10] ;%{PE}
;FOLD Parameters ;%{h}
;Params IlfProvider=kukaroboter.basistech.inlineforms.movement.old; Kuka.IsGlobalPoint=False; Kuka.PointName=P42; Kuka.BlendingEnabled=TRUE; Kuka.MoveDataName=CPDATP42; Kuka.VelocityPath=1; Kuka.CurrentCDSetIndex=0; Kuka.MovementParameterFieldEnabled=True; IlfCommand=LIN
;ENDFOLD
$BWDSTART = FALSE
LDAT_ACT=LCPDATP42
FDAT_ACT=FP42
BAS (#CP_PARAMS,1)
SET_CD_PARAMS (0)
LIN XP42 C_DIS

;ENDFOLD
;FOLD LIN P43 CONT Vel=1 m/s CPDATP43 Tool[2] Base[10] ;%{PE}
;FOLD Parameters ;%{h}
;Params IlfProvider=kukaroboter.basistech.inlineforms.movement.old; Kuka.IsGlobalPoint=False; Kuka.PointName=P43; Kuka.BlendingEnabled=TRUE; Kuka.MoveDataName=CPDATP43; Kuka.VelocityPath=1; Kuka.CurrentCDSetIndex=0; Kuka.MovementParameterFieldEnabled=True; IlfCommand=LIN
;ENDFOLD
$BWDSTART = FALSE
LDAT_ACT=LCPDATP43
FDAT_ACT=FP43
BAS (#CP_PARAMS,1)
SET_CD_PARAMS (0)
LIN XP43 C_DIS

;ENDFOLD
;FOLD CIRC CAux44 CDes44 CONT Vel=0.1 m/s CPDATC44 Tool[2] Base[10] ;%{PE}
;FOLD Parameters ;%{h}
;Params IlfProvider=kukaroboter.basistech.inlineforms.movement.old; Kuka.IsGlobalPoint=False; Kuka.PointName=CDes44; Kuka.BlendingEnabled=TRUE; Kuka.MoveDataName=CPDATC44; Kuka.VelocityPath=0.1; Kuka.CurrentCDSetIndex=0; Kuka.MovementParameterFieldEnabled=True; IlfCommand=LIN
;ENDFOLD
$BWDSTART = FALSE
LDAT_ACT=LCPDATC44
FDAT_ACT=FC44
$ORI_TYPE = #VAR
$CIRC_TYPE = #PATH
BAS (#CP_PARAMS,0.1)
SET_CD_PARAMS (0)
CIRC XCAux44, XCDes44 C_DIS

;ENDFOLD
;FOLD LIN P45 CONT Vel=1 m/s CPDATP45 Tool[2] Base[10] ;%{PE}
;FOLD Parameters ;%{h}
;Params IlfProvider=kukaroboter.basistech.inlineforms.movement.old; Kuka.IsGlobalPoint=False; Kuka.PointName=P45; Kuka.BlendingEnabled=TRUE; Kuka.MoveDataName=CPDATP45; Kuka.VelocityPath=1; Kuka.CurrentCDSetIndex=0; Kuka.MovementParameterFieldEnabled=True; IlfCommand=LIN
;ENDFOLD
$BWDSTART = FALSE
LDAT_ACT=LCPDATP45
FDAT_ACT=FP45
BAS (#CP_PARAMS,1)
SET_CD_PARAMS (0)
LIN XP45 C_DIS

;ENDFOLD
;FOLD LIN P46 CONT Vel=1 m/s CPDATP46 Tool[2] Base[10] ;%{PE}
;FOLD Parameters ;%{h}
;Params IlfProvider=kukaroboter.basistech.inlineforms.movement.old; Kuka.IsGlobalPoint=False; Kuka.PointName=P46; Kuka.BlendingEnabled=TRUE; Kuka.MoveDataName=CPDATP46; Kuka.VelocityPath=1; Kuka.CurrentCDSetIndex=0; Kuka.MovementParameterFieldEnabled=True; IlfCommand=LIN
;ENDFOLD
$BWDSTART = FALSE
LDAT_ACT=LCPDATP46
FDAT_ACT=FP46
BAS (#CP_PARAMS,1)
SET_CD_PARAMS (0)
LIN XP46 C_DIS

;ENDFOLD
;FOLD CIRC CAux47 CDes47 CONT Vel=0.1 m/s CPDATC47 Tool[2] Base[10] ;%{PE}
;FOLD Parameters ;%{h}
;Params IlfProvider=kukaroboter.basistech.inlineforms.movement.old; Kuka.IsGlobalPoint=False; Kuka.PointName=CDes47; Kuka.BlendingEnabled=TRUE; Kuka.MoveDataName=CPDATC47; Kuka.VelocityPath=0.1; Kuka.CurrentCDSetIndex=0; Kuka.MovementParameterFieldEnabled=True; IlfCommand=LIN
;ENDFOLD
$BWDSTART = FALSE
LDAT_ACT=LCPDATC47
FDAT_ACT=FC47
$ORI_TYPE = #VAR
$CIRC_TYPE = #PATH
BAS (#CP_PARAMS,0.1)
SET_CD_PARAMS (0)
CIRC XCAux47, XCDes47 C_DIS

;ENDFOLD
;FOLD LIN P48 CONT Vel=1 m/s CPDATP48 Tool[2] Base[10] ;%{PE}
;FOLD Parameters ;%{h}
;Params IlfProvider=kukaroboter.basistech.inlineforms.movement.old; Kuka.IsGlobalPoint=False; Kuka.PointName=P48; Kuka.BlendingEnabled=TRUE; Kuka.MoveDataName=CPDATP48; Kuka.VelocityPath=1; Kuka.CurrentCDSetIndex=0; Kuka.MovementParameterFieldEnabled=True; IlfCommand=LIN
;ENDFOLD
$BWDSTART = FALSE
LDAT_ACT=LCPDATP48
FDAT_ACT=FP48
BAS (#CP_PARAMS,1)
SET_CD_PARAMS (0)
LIN XP48 C_DIS

;ENDFOLD
;FOLD LIN P49 CONT Vel=1 m/s CPDATP49 Tool[2] Base[10] ;%{PE}
;FOLD Parameters ;%{h}
;Params IlfProvider=kukaroboter.basistech.inlineforms.movement.old; Kuka.IsGlobalPoint=False; Kuka.PointName=P49; Kuka.BlendingEnabled=TRUE; Kuka.MoveDataName=CPDATP49; Kuka.VelocityPath=1; Kuka.CurrentCDSetIndex=0; Kuka.MovementParameterFieldEnabled=True; IlfCommand=LIN
;ENDFOLD
$BWDSTART = FALSE
LDAT_ACT=LCPDATP49
FDAT_ACT=FP49
BAS (#CP_PARAMS,1)
SET_CD_PARAMS (0)
LIN XP49 C_DIS

;ENDFOLD
;FOLD CIRC CAux50 CDes50 CONT Vel=0.1 m/s CPDATC50 Tool[2] Base[10] ;%{PE}
;FOLD Parameters ;%{h}
;Params IlfProvider=kukaroboter.basistech.inlineforms.movement.old; Kuka.IsGlobalPoint=False; Kuka.PointName=CDes50; Kuka.BlendingEnabled=TRUE; Kuka.MoveDataName=CPDATC50; Kuka.VelocityPath=0.1; Kuka.CurrentCDSetIndex=0; Kuka.MovementParameterFieldEnabled=True; IlfCommand=LIN
;ENDFOLD
$BWDSTART = FALSE
LDAT_ACT=LCPDATC50
FDAT_ACT=FC50
$ORI_TYPE = #VAR
$CIRC_TYPE = #PATH
BAS (#CP_PARAMS,0.1)
SET_CD_PARAMS (0)
CIRC XCAux50, XCDes50 C_DIS

;ENDFOLD
;FOLD LIN P51 CONT Vel=1 m/s CPDATP51 Tool[2] Base[10] ;%{PE}
;FOLD Parameters ;%{h}
;Params IlfProvider=kukaroboter.basistech.inlineforms.movement.old; Kuka.IsGlobalPoint=False; Kuka.PointName=P51; Kuka.BlendingEnabled=TRUE; Kuka.MoveDataName=CPDATP51; Kuka.VelocityPath=1; Kuka.CurrentCDSetIndex=0; Kuka.MovementParameterFieldEnabled=True; IlfCommand=LIN
;ENDFOLD
$BWDSTART = FALSE
LDAT_ACT=LCPDATP51
FDAT_ACT=FP51
BAS (#CP_PARAMS,1)
SET_CD_PARAMS (0)
LIN XP51 C_DIS

;ENDFOLD
;FOLD LIN P52 CONT Vel=1 m/s CPDATP52 Tool[2] Base[10] ;%{PE}
;FOLD Parameters ;%{h}
;Params IlfProvider=kukaroboter.basistech.inlineforms.movement.old; Kuka.IsGlobalPoint=False; Kuka.PointName=P52; Kuka.BlendingEnabled=TRUE; Kuka.MoveDataName=CPDATP52; Kuka.VelocityPath=1; Kuka.CurrentCDSetIndex=0; Kuka.MovementParameterFieldEnabled=True; IlfCommand=LIN
;ENDFOLD
$BWDSTART = FALSE
LDAT_ACT=LCPDATP52
FDAT_ACT=FP52
BAS (#CP_PARAMS,1)
SET_CD_PARAMS (0)
LIN XP52 C_DIS

;ENDFOLD
;FOLD CIRC CAux53 CDes53 CONT Vel=0.1 m/s CPDATC53 Tool[2] Base[10] ;%{PE}
;FOLD Parameters ;%{h}
;Params IlfProvider=kukaroboter.basistech.inlineforms.movement.old; Kuka.IsGlobalPoint=False; Kuka.PointName=CDes53; Kuka.BlendingEnabled=TRUE; Kuka.MoveDataName=CPDATC53; Kuka.VelocityPath=0.1; Kuka.CurrentCDSetIndex=0; Kuka.MovementParameterFieldEnabled=True; IlfCommand=LIN
;ENDFOLD
$BWDSTART = FALSE
LDAT_ACT=LCPDATC53
FDAT_ACT=FC53
$ORI_TYPE = #VAR
$CIRC_TYPE = #PATH
BAS (#CP_PARAMS,0.1)
SET_CD_PARAMS (0)
CIRC XCAux53, XCDes53 C_DIS

;ENDFOLD
;FOLD LIN P54 CONT Vel=1 m/s CPDATP54 Tool[2] Base[10] ;%{PE}
;FOLD Parameters ;%{h}
;Params IlfProvider=kukaroboter.basistech.inlineforms.movement.old; Kuka.IsGlobalPoint=False; Kuka.PointName=P54; Kuka.BlendingEnabled=TRUE; Kuka.MoveDataName=CPDATP54; Kuka.VelocityPath=1; Kuka.CurrentCDSetIndex=0; Kuka.MovementParameterFieldEnabled=True; IlfCommand=LIN
;ENDFOLD
$BWDSTART = FALSE
LDAT_ACT=LCPDATP54
FDAT_ACT=FP54
BAS (#CP_PARAMS,1)
SET_CD_PARAMS (0)
LIN XP54 C_DIS

;ENDFOLD
;FOLD LIN P55 CONT Vel=1 m/s CPDATP55 Tool[2] Base[10] ;%{PE}
;FOLD Parameters ;%{h}
;Params IlfProvider=kukaroboter.basistech.inlineforms.movement.old; Kuka.IsGlobalPoint=False; Kuka.PointName=P55; Kuka.BlendingEnabled=TRUE; Kuka.MoveDataName=CPDATP55; Kuka.VelocityPath=1; Kuka.CurrentCDSetIndex=0; Kuka.MovementParameterFieldEnabled=True; IlfCommand=LIN
;ENDFOLD
$BWDSTART = FALSE
LDAT_ACT=LCPDATP55
FDAT_ACT=FP55
BAS (#CP_PARAMS,1)
SET_CD_PARAMS (0)
LIN XP55 C_DIS

;ENDFOLD
;FOLD CIRC CAux56 CDes56 CONT Vel=0.1 m/s CPDATC56 Tool[2] Base[10] ;%{PE}
;FOLD Parameters ;%{h}
;Params IlfProvider=kukaroboter.basistech.inlineforms.movement.old; Kuka.IsGlobalPoint=False; Kuka.PointName=CDes56; Kuka.BlendingEnabled=TRUE; Kuka.MoveDataName=CPDATC56; Kuka.VelocityPath=0.1; Kuka.CurrentCDSetIndex=0; Kuka.MovementParameterFieldEnabled=True; IlfCommand=LIN
;ENDFOLD
$BWDSTART = FALSE
LDAT_ACT=LCPDATC56
FDAT_ACT=FC56
$ORI_TYPE = #VAR
$CIRC_TYPE = #PATH
BAS (#CP_PARAMS,0.1)
SET_CD_PARAMS (0)
CIRC XCAux56, XCDes56 C_DIS

;ENDFOLD
;FOLD LIN P57 CONT Vel=1 m/s CPDATP57 Tool[2] Base[10] ;%{PE}
;FOLD Parameters ;%{h}
;Params IlfProvider=kukaroboter.basistech.inlineforms.movement.old; Kuka.IsGlobalPoint=False; Kuka.PointName=P57; Kuka.BlendingEnabled=TRUE; Kuka.MoveDataName=CPDATP57; Kuka.VelocityPath=1; Kuka.CurrentCDSetIndex=0; Kuka.MovementParameterFieldEnabled=True; IlfCommand=LIN
;ENDFOLD
$BWDSTART = FALSE
LDAT_ACT=LCPDATP57
FDAT_ACT=FP57
BAS (#CP_PARAMS,1)
SET_CD_PARAMS (0)
LIN XP57 C_DIS

;ENDFOLD
;FOLD LIN P58 CONT Vel=1 m/s CPDATP58 Tool[2] Base[10] ;%{PE}
;FOLD Parameters ;%{h}
;Params IlfProvider=kukaroboter.basistech.inlineforms.movement.old; Kuka.IsGlobalPoint=False; Kuka.PointName=P58; Kuka.BlendingEnabled=TRUE; Kuka.MoveDataName=CPDATP58; Kuka.VelocityPath=1; Kuka.CurrentCDSetIndex=0; Kuka.MovementParameterFieldEnabled=True; IlfCommand=LIN
;ENDFOLD
$BWDSTART = FALSE
LDAT_ACT=LCPDATP58
FDAT_ACT=FP58
BAS (#CP_PARAMS,1)
SET_CD_PARAMS (0)
LIN XP58 C_DIS

;ENDFOLD
;FOLD CIRC CAux59 CDes59 CONT Vel=0.1 m/s CPDATC59 Tool[2] Base[10] ;%{PE}
;FOLD Parameters ;%{h}
;Params IlfProvider=kukaroboter.basistech.inlineforms.movement.old; Kuka.IsGlobalPoint=False; Kuka.PointName=CDes59; Kuka.BlendingEnabled=TRUE; Kuka.MoveDataName=CPDATC59; Kuka.VelocityPath=0.1; Kuka.CurrentCDSetIndex=0; Kuka.MovementParameterFieldEnabled=True; IlfCommand=LIN
;ENDFOLD
$BWDSTART = FALSE
LDAT_ACT=LCPDATC59
FDAT_ACT=FC59
$ORI_TYPE = #VAR
$CIRC_TYPE = #PATH
BAS (#CP_PARAMS,0.1)
SET_CD_PARAMS (0)
CIRC XCAux59, XCDes59 C_DIS

;ENDFOLD
;FOLD LIN P60 CONT Vel=1 m/s CPDATP60 Tool[2] Base[10] ;%{PE}
;FOLD Parameters ;%{h}
;Params IlfProvider=kukaroboter.basistech.inlineforms.movement.old; Kuka.IsGlobalPoint=False; Kuka.PointName=P60; Kuka.BlendingEnabled=TRUE; Kuka.MoveDataName=CPDATP60; Kuka.VelocityPath=1; Kuka.CurrentCDSetIndex=0; Kuka.MovementParameterFieldEnabled=True; IlfCommand=LIN
;ENDFOLD
$BWDSTART = FALSE
LDAT_ACT=LCPDATP60
FDAT_ACT=FP60
BAS (#CP_PARAMS,1)
SET_CD_PARAMS (0)
LIN XP60 C_DIS

;ENDFOLD
;FOLD LIN P61 CONT Vel=1 m/s CPDATP61 Tool[2] Base[10] ;%{PE}
;FOLD Parameters ;%{h}
;Params IlfProvider=kukaroboter.basistech.inlineforms.movement.old; Kuka.IsGlobalPoint=False; Kuka.PointName=P61; Kuka.BlendingEnabled=TRUE; Kuka.MoveDataName=CPDATP61; Kuka.VelocityPath=1; Kuka.CurrentCDSetIndex=0; Kuka.MovementParameterFieldEnabled=True; IlfCommand=LIN
;ENDFOLD
$BWDSTART = FALSE
LDAT_ACT=LCPDATP61
FDAT_ACT=FP61
BAS (#CP_PARAMS,1)
SET_CD_PARAMS (0)
LIN XP61 C_DIS

;ENDFOLD
;FOLD CIRC CAux62 CDes62 CONT Vel=0.1 m/s CPDATC62 Tool[2] Base[10] ;%{PE}
;FOLD Parameters ;%{h}
;Params IlfProvider=kukaroboter.basistech.inlineforms.movement.old; Kuka.IsGlobalPoint=False; Kuka.PointName=CDes62; Kuka.BlendingEnabled=TRUE; Kuka.MoveDataName=CPDATC62; Kuka.VelocityPath=0.1; Kuka.CurrentCDSetIndex=0; Kuka.MovementParameterFieldEnabled=True; IlfCommand=LIN
;ENDFOLD
$BWDSTART = FALSE
LDAT_ACT=LCPDATC62
FDAT_ACT=FC62
$ORI_TYPE = #VAR
$CIRC_TYPE = #PATH
BAS (#CP_PARAMS,0.1)
SET_CD_PARAMS (0)
CIRC XCAux62, XCDes62 C_DIS

;ENDFOLD
;FOLD LIN P63 CONT Vel=1 m/s CPDATP63 Tool[2] Base[10] ;%{PE}
;FOLD Parameters ;%{h}
;Params IlfProvider=kukaroboter.basistech.inlineforms.movement.old; Kuka.IsGlobalPoint=False; Kuka.PointName=P63; Kuka.BlendingEnabled=TRUE; Kuka.MoveDataName=CPDATP63; Kuka.VelocityPath=1; Kuka.CurrentCDSetIndex=0; Kuka.MovementParameterFieldEnabled=True; IlfCommand=LIN
;ENDFOLD
$BWDSTART = FALSE
LDAT_ACT=LCPDATP63
FDAT_ACT=FP63
BAS (#CP_PARAMS,1)
SET_CD_PARAMS (0)
LIN XP63 C_DIS

;ENDFOLD
;FOLD LIN P64 CONT Vel=1 m/s CPDATP64 Tool[2] Base[10] ;%{PE}
;FOLD Parameters ;%{h}
;Params IlfProvider=kukaroboter.basistech.inlineforms.movement.old; Kuka.IsGlobalPoint=False; Kuka.PointName=P64; Kuka.BlendingEnabled=TRUE; Kuka.MoveDataName=CPDATP64; Kuka.VelocityPath=1; Kuka.CurrentCDSetIndex=0; Kuka.MovementParameterFieldEnabled=True; IlfCommand=LIN
;ENDFOLD
$BWDSTART = FALSE
LDAT_ACT=LCPDATP64
FDAT_ACT=FP64
BAS (#CP_PARAMS,1)
SET_CD_PARAMS (0)
LIN XP64 C_DIS

;ENDFOLD
;FOLD CIRC CAux65 CDes65 CONT Vel=0.1 m/s CPDATC65 Tool[2] Base[10] ;%{PE}
;FOLD Parameters ;%{h}
;Params IlfProvider=kukaroboter.basistech.inlineforms.movement.old; Kuka.IsGlobalPoint=False; Kuka.PointName=CDes65; Kuka.BlendingEnabled=TRUE; Kuka.MoveDataName=CPDATC65; Kuka.VelocityPath=0.1; Kuka.CurrentCDSetIndex=0; Kuka.MovementParameterFieldEnabled=True; IlfCommand=LIN
;ENDFOLD
$BWDSTART = FALSE
LDAT_ACT=LCPDATC65
FDAT_ACT=FC65
$ORI_TYPE = #VAR
$CIRC_TYPE = #PATH
BAS (#CP_PARAMS,0.1)
SET_CD_PARAMS (0)
CIRC XCAux65, XCDes65 C_DIS

;ENDFOLD
;FOLD LIN P66 CONT Vel=1 m/s CPDATP66 Tool[2] Base[10] ;%{PE}
;FOLD Parameters ;%{h}
;Params IlfProvider=kukaroboter.basistech.inlineforms.movement.old; Kuka.IsGlobalPoint=False; Kuka.PointName=P66; Kuka.BlendingEnabled=TRUE; Kuka.MoveDataName=CPDATP66; Kuka.VelocityPath=1; Kuka.CurrentCDSetIndex=0; Kuka.MovementParameterFieldEnabled=True; IlfCommand=LIN
;ENDFOLD
$BWDSTART = FALSE
LDAT_ACT=LCPDATP66
FDAT_ACT=FP66
BAS (#CP_PARAMS,1)
SET_CD_PARAMS (0)
LIN XP66 C_DIS

;ENDFOLD
;FOLD LIN P67 CONT Vel=1 m/s CPDATP67 Tool[2] Base[10] ;%{PE}
;FOLD Parameters ;%{h}
;Params IlfProvider=kukaroboter.basistech.inlineforms.movement.old; Kuka.IsGlobalPoint=False; Kuka.PointName=P67; Kuka.BlendingEnabled=TRUE; Kuka.MoveDataName=CPDATP67; Kuka.VelocityPath=1; Kuka.CurrentCDSetIndex=0; Kuka.MovementParameterFieldEnabled=True; IlfCommand=LIN
;ENDFOLD
$BWDSTART = FALSE
LDAT_ACT=LCPDATP67
FDAT_ACT=FP67
BAS (#CP_PARAMS,1)
SET_CD_PARAMS (0)
LIN XP67 C_DIS

;ENDFOLD
;FOLD CIRC CAux68 CDes68 CONT Vel=0.1 m/s CPDATC68 Tool[2] Base[10] ;%{PE}
;FOLD Parameters ;%{h}
;Params IlfProvider=kukaroboter.basistech.inlineforms.movement.old; Kuka.IsGlobalPoint=False; Kuka.PointName=CDes68; Kuka.BlendingEnabled=TRUE; Kuka.MoveDataName=CPDATC68; Kuka.VelocityPath=0.1; Kuka.CurrentCDSetIndex=0; Kuka.MovementParameterFieldEnabled=True; IlfCommand=LIN
;ENDFOLD
$BWDSTART = FALSE
LDAT_ACT=LCPDATC68
FDAT_ACT=FC68
$ORI_TYPE = #VAR
$CIRC_TYPE = #PATH
BAS (#CP_PARAMS,0.1)
SET_CD_PARAMS (0)
CIRC XCAux68, XCDes68 C_DIS

;ENDFOLD
;FOLD LIN P69 CONT Vel=1 m/s CPDATP69 Tool[2] Base[10] ;%{PE}
;FOLD Parameters ;%{h}
;Params IlfProvider=kukaroboter.basistech.inlineforms.movement.old; Kuka.IsGlobalPoint=False; Kuka.PointName=P69; Kuka.BlendingEnabled=TRUE; Kuka.MoveDataName=CPDATP69; Kuka.VelocityPath=1; Kuka.CurrentCDSetIndex=0; Kuka.MovementParameterFieldEnabled=True; IlfCommand=LIN
;ENDFOLD
$BWDSTART = FALSE
LDAT_ACT=LCPDATP69
FDAT_ACT=FP69
BAS (#CP_PARAMS,1)
SET_CD_PARAMS (0)
LIN XP69 C_DIS

;ENDFOLD
;FOLD LIN P70 CONT Vel=1 m/s CPDATP70 Tool[2] Base[10] ;%{PE}
;FOLD Parameters ;%{h}
;Params IlfProvider=kukaroboter.basistech.inlineforms.movement.old; Kuka.IsGlobalPoint=False; Kuka.PointName=P70; Kuka.BlendingEnabled=TRUE; Kuka.MoveDataName=CPDATP70; Kuka.VelocityPath=1; Kuka.CurrentCDSetIndex=0; Kuka.MovementParameterFieldEnabled=True; IlfCommand=LIN
;ENDFOLD
$BWDSTART = FALSE
LDAT_ACT=LCPDATP70
FDAT_ACT=FP70
BAS (#CP_PARAMS,1)
SET_CD_PARAMS (0)
LIN XP70 C_DIS

;ENDFOLD
;FOLD CIRC CAux71 CDes71 CONT Vel=0.1 m/s CPDATC71 Tool[2] Base[10] ;%{PE}
;FOLD Parameters ;%{h}
;Params IlfProvider=kukaroboter.basistech.inlineforms.movement.old; Kuka.IsGlobalPoint=False; Kuka.PointName=CDes71; Kuka.BlendingEnabled=TRUE; Kuka.MoveDataName=CPDATC71; Kuka.VelocityPath=0.1; Kuka.CurrentCDSetIndex=0; Kuka.MovementParameterFieldEnabled=True; IlfCommand=LIN
;ENDFOLD
$BWDSTART = FALSE
LDAT_ACT=LCPDATC71
FDAT_ACT=FC71
$ORI_TYPE = #VAR
$CIRC_TYPE = #PATH
BAS (#CP_PARAMS,0.1)
SET_CD_PARAMS (0)
CIRC XCAux71, XCDes71 C_DIS

;ENDFOLD
;FOLD LIN P72 CONT Vel=1 m/s CPDATP72 Tool[2] Base[10] ;%{PE}
;FOLD Parameters ;%{h}
;Params IlfProvider=kukaroboter.basistech.inlineforms.movement.old; Kuka.IsGlobalPoint=False; Kuka.PointName=P72; Kuka.BlendingEnabled=TRUE; Kuka.MoveDataName=CPDATP72; Kuka.VelocityPath=1; Kuka.CurrentCDSetIndex=0; Kuka.MovementParameterFieldEnabled=True; IlfCommand=LIN
;ENDFOLD
$BWDSTART = FALSE
LDAT_ACT=LCPDATP72
FDAT_ACT=FP72
BAS (#CP_PARAMS,1)
SET_CD_PARAMS (0)
LIN XP72 C_DIS

;ENDFOLD
;FOLD LIN P73 CONT Vel=1 m/s CPDATP73 Tool[2] Base[10] ;%{PE}
;FOLD Parameters ;%{h}
;Params IlfProvider=kukaroboter.basistech.inlineforms.movement.old; Kuka.IsGlobalPoint=False; Kuka.PointName=P73; Kuka.BlendingEnabled=TRUE; Kuka.MoveDataName=CPDATP73; Kuka.VelocityPath=1; Kuka.CurrentCDSetIndex=0; Kuka.MovementParameterFieldEnabled=True; IlfCommand=LIN
;ENDFOLD
$BWDSTART = FALSE
LDAT_ACT=LCPDATP73
FDAT_ACT=FP73
BAS (#CP_PARAMS,1)
SET_CD_PARAMS (0)
LIN XP73 C_DIS

;ENDFOLD
;FOLD CIRC CAux74 CDes74 CONT Vel=0.1 m/s CPDATC74 Tool[2] Base[10] ;%{PE}
;FOLD Parameters ;%{h}
;Params IlfProvider=kukaroboter.basistech.inlineforms.movement.old; Kuka.IsGlobalPoint=False; Kuka.PointName=CDes74; Kuka.BlendingEnabled=TRUE; Kuka.MoveDataName=CPDATC74; Kuka.VelocityPath=0.1; Kuka.CurrentCDSetIndex=0; Kuka.MovementParameterFieldEnabled=True; IlfCommand=LIN
;ENDFOLD
$BWDSTART = FALSE
LDAT_ACT=LCPDATC74
FDAT_ACT=FC74
$ORI_TYPE = #VAR
$CIRC_TYPE = #PATH
BAS (#CP_PARAMS,0.1)
SET_CD_PARAMS (0)
CIRC XCAux74, XCDes74 C_DIS

;ENDFOLD
;FOLD LIN P75 CONT Vel=1 m/s CPDATP75 Tool[2] Base[10] ;%{PE}
;FOLD Parameters ;%{h}
;Params IlfProvider=kukaroboter.basistech.inlineforms.movement.old; Kuka.IsGlobalPoint=False; Kuka.PointName=P75; Kuka.BlendingEnabled=TRUE; Kuka.MoveDataName=CPDATP75; Kuka.VelocityPath=1; Kuka.CurrentCDSetIndex=0; Kuka.MovementParameterFieldEnabled=True; IlfCommand=LIN
;ENDFOLD
$BWDSTART = FALSE
LDAT_ACT=LCPDATP75
FDAT_ACT=FP75
BAS (#CP_PARAMS,1)
SET_CD_PARAMS (0)
LIN XP75 C_DIS

;ENDFOLD
;FOLD LIN P76 CONT Vel=1 m/s CPDATP76 Tool[2] Base[10] ;%{PE}
;FOLD Parameters ;%{h}
;Params IlfProvider=kukaroboter.basistech.inlineforms.movement.old; Kuka.IsGlobalPoint=False; Kuka.PointName=P76; Kuka.BlendingEnabled=TRUE; Kuka.MoveDataName=CPDATP76; Kuka.VelocityPath=1; Kuka.CurrentCDSetIndex=0; Kuka.MovementParameterFieldEnabled=True; IlfCommand=LIN
;ENDFOLD
$BWDSTART = FALSE
LDAT_ACT=LCPDATP76
FDAT_ACT=FP76
BAS (#CP_PARAMS,1)
SET_CD_PARAMS (0)
LIN XP76 C_DIS

;ENDFOLD
;FOLD CIRC CAux77 CDes77 CONT Vel=0.1 m/s CPDATC77 Tool[2] Base[10] ;%{PE}
;FOLD Parameters ;%{h}
;Params IlfProvider=kukaroboter.basistech.inlineforms.movement.old; Kuka.IsGlobalPoint=False; Kuka.PointName=CDes77; Kuka.BlendingEnabled=TRUE; Kuka.MoveDataName=CPDATC77; Kuka.VelocityPath=0.1; Kuka.CurrentCDSetIndex=0; Kuka.MovementParameterFieldEnabled=True; IlfCommand=LIN
;ENDFOLD
$BWDSTART = FALSE
LDAT_ACT=LCPDATC77
FDAT_ACT=FC77
$ORI_TYPE = #VAR
$CIRC_TYPE = #PATH
BAS (#CP_PARAMS,0.1)
SET_CD_PARAMS (0)
CIRC XCAux77, XCDes77 C_DIS

;ENDFOLD
;FOLD LIN P78 CONT Vel=1 m/s CPDATP78 Tool[2] Base[10] ;%{PE}
;FOLD Parameters ;%{h}
;Params IlfProvider=kukaroboter.basistech.inlineforms.movement.old; Kuka.IsGlobalPoint=False; Kuka.PointName=P78; Kuka.BlendingEnabled=TRUE; Kuka.MoveDataName=CPDATP78; Kuka.VelocityPath=1; Kuka.CurrentCDSetIndex=0; Kuka.MovementParameterFieldEnabled=True; IlfCommand=LIN
;ENDFOLD
$BWDSTART = FALSE
LDAT_ACT=LCPDATP78
FDAT_ACT=FP78
BAS (#CP_PARAMS,1)
SET_CD_PARAMS (0)
LIN XP78 C_DIS

;ENDFOLD
;FOLD LIN P79 CONT Vel=1 m/s CPDATP79 Tool[2] Base[10] ;%{PE}
;FOLD Parameters ;%{h}
;Params IlfProvider=kukaroboter.basistech.inlineforms.movement.old; Kuka.IsGlobalPoint=False; Kuka.PointName=P79; Kuka.BlendingEnabled=TRUE; Kuka.MoveDataName=CPDATP79; Kuka.VelocityPath=1; Kuka.CurrentCDSetIndex=0; Kuka.MovementParameterFieldEnabled=True; IlfCommand=LIN
;ENDFOLD
$BWDSTART = FALSE
LDAT_ACT=LCPDATP79
FDAT_ACT=FP79
BAS (#CP_PARAMS,1)
SET_CD_PARAMS (0)
LIN XP79 C_DIS

;ENDFOLD
;FOLD CIRC CAux80 CDes80 CONT Vel=0.1 m/s CPDATC80 Tool[2] Base[10] ;%{PE}
;FOLD Parameters ;%{h}
;Params IlfProvider=kukaroboter.basistech.inlineforms.movement.old; Kuka.IsGlobalPoint=False; Kuka.PointName=CDes80; Kuka.BlendingEnabled=TRUE; Kuka.MoveDataName=CPDATC80; Kuka.VelocityPath=0.1; Kuka.CurrentCDSetIndex=0; Kuka.MovementParameterFieldEnabled=True; IlfCommand=LIN
;ENDFOLD
$BWDSTART = FALSE
LDAT_ACT=LCPDATC80
FDAT_ACT=FC80
$ORI_TYPE = #VAR
$CIRC_TYPE = #PATH
BAS (#CP_PARAMS,0.1)
SET_CD_PARAMS (0)
CIRC XCAux80, XCDes80 C_DIS

;ENDFOLD
;FOLD LIN P81 CONT Vel=1 m/s CPDATP81 Tool[2] Base[10] ;%{PE}
;FOLD Parameters ;%{h}
;Params IlfProvider=kukaroboter.basistech.inlineforms.movement.old; Kuka.IsGlobalPoint=False; Kuka.PointName=P81; Kuka.BlendingEnabled=TRUE; Kuka.MoveDataName=CPDATP81; Kuka.VelocityPath=1; Kuka.CurrentCDSetIndex=0; Kuka.MovementParameterFieldEnabled=True; IlfCommand=LIN
;ENDFOLD
$BWDSTART = FALSE
LDAT_ACT=LCPDATP81
FDAT_ACT=FP81
BAS (#CP_PARAMS,1)
SET_CD_PARAMS (0)
LIN XP81 C_DIS

;ENDFOLD
;FOLD LIN P82 CONT Vel=1 m/s CPDATP82 Tool[2] Base[10] ;%{PE}
;FOLD Parameters ;%{h}
;Params IlfProvider=kukaroboter.basistech.inlineforms.movement.old; Kuka.IsGlobalPoint=False; Kuka.PointName=P82; Kuka.BlendingEnabled=TRUE; Kuka.MoveDataName=CPDATP82; Kuka.VelocityPath=1; Kuka.CurrentCDSetIndex=0; Kuka.MovementParameterFieldEnabled=True; IlfCommand=LIN
;ENDFOLD
$BWDSTART = FALSE
LDAT_ACT=LCPDATP82
FDAT_ACT=FP82
BAS (#CP_PARAMS,1)
SET_CD_PARAMS (0)
LIN XP82 C_DIS

;ENDFOLD
;FOLD CIRC CAux83 CDes83 CONT Vel=0.1 m/s CPDATC83 Tool[2] Base[10] ;%{PE}
;FOLD Parameters ;%{h}
;Params IlfProvider=kukaroboter.basistech.inlineforms.movement.old; Kuka.IsGlobalPoint=False; Kuka.PointName=CDes83; Kuka.BlendingEnabled=TRUE; Kuka.MoveDataName=CPDATC83; Kuka.VelocityPath=0.1; Kuka.CurrentCDSetIndex=0; Kuka.MovementParameterFieldEnabled=True; IlfCommand=LIN
;ENDFOLD
$BWDSTART = FALSE
LDAT_ACT=LCPDATC83
FDAT_ACT=FC83
$ORI_TYPE = #VAR
$CIRC_TYPE = #PATH
BAS (#CP_PARAMS,0.1)
SET_CD_PARAMS (0)
CIRC XCAux83, XCDes83 C_DIS

;ENDFOLD
;FOLD LIN P84 CONT Vel=1 m/s CPDATP84 Tool[2] Base[10] ;%{PE}
;FOLD Parameters ;%{h}
;Params IlfProvider=kukaroboter.basistech.inlineforms.movement.old; Kuka.IsGlobalPoint=False; Kuka.PointName=P84; Kuka.BlendingEnabled=TRUE; Kuka.MoveDataName=CPDATP84; Kuka.VelocityPath=1; Kuka.CurrentCDSetIndex=0; Kuka.MovementParameterFieldEnabled=True; IlfCommand=LIN
;ENDFOLD
$BWDSTART = FALSE
LDAT_ACT=LCPDATP84
FDAT_ACT=FP84
BAS (#CP_PARAMS,1)
SET_CD_PARAMS (0)
LIN XP84 C_DIS

;ENDFOLD
;FOLD LIN P85 CONT Vel=1 m/s CPDATP85 Tool[2] Base[10] ;%{PE}
;FOLD Parameters ;%{h}
;Params IlfProvider=kukaroboter.basistech.inlineforms.movement.old; Kuka.IsGlobalPoint=False; Kuka.PointName=P85; Kuka.BlendingEnabled=TRUE; Kuka.MoveDataName=CPDATP85; Kuka.VelocityPath=1; Kuka.CurrentCDSetIndex=0; Kuka.MovementParameterFieldEnabled=True; IlfCommand=LIN
;ENDFOLD
$BWDSTART = FALSE
LDAT_ACT=LCPDATP85
FDAT_ACT=FP85
BAS (#CP_PARAMS,1)
SET_CD_PARAMS (0)
LIN XP85 C_DIS

;ENDFOLD
;FOLD CIRC CAux86 CDes86 CONT Vel=0.1 m/s CPDATC86 Tool[2] Base[10] ;%{PE}
;FOLD Parameters ;%{h}
;Params IlfProvider=kukaroboter.basistech.inlineforms.movement.old; Kuka.IsGlobalPoint=False; Kuka.PointName=CDes86; Kuka.BlendingEnabled=TRUE; Kuka.MoveDataName=CPDATC86; Kuka.VelocityPath=0.1; Kuka.CurrentCDSetIndex=0; Kuka.MovementParameterFieldEnabled=True; IlfCommand=LIN
;ENDFOLD
$BWDSTART = FALSE
LDAT_ACT=LCPDATC86
FDAT_ACT=FC86
$ORI_TYPE = #VAR
$CIRC_TYPE = #PATH
BAS (#CP_PARAMS,0.1)
SET_CD_PARAMS (0)
CIRC XCAux86, XCDes86 C_DIS

;ENDFOLD
;FOLD LIN P87 CONT Vel=1 m/s CPDATP87 Tool[2] Base[10] ;%{PE}
;FOLD Parameters ;%{h}
;Params IlfProvider=kukaroboter.basistech.inlineforms.movement.old; Kuka.IsGlobalPoint=False; Kuka.PointName=P87; Kuka.BlendingEnabled=TRUE; Kuka.MoveDataName=CPDATP87; Kuka.VelocityPath=1; Kuka.CurrentCDSetIndex=0; Kuka.MovementParameterFieldEnabled=True; IlfCommand=LIN
;ENDFOLD
$BWDSTART = FALSE
LDAT_ACT=LCPDATP87
FDAT_ACT=FP87
BAS (#CP_PARAMS,1)
SET_CD_PARAMS (0)
LIN XP87 C_DIS

;ENDFOLD
;FOLD LIN P88 CONT Vel=1 m/s CPDATP88 Tool[2] Base[10] ;%{PE}
;FOLD Parameters ;%{h}
;Params IlfProvider=kukaroboter.basistech.inlineforms.movement.old; Kuka.IsGlobalPoint=False; Kuka.PointName=P88; Kuka.BlendingEnabled=TRUE; Kuka.MoveDataName=CPDATP88; Kuka.VelocityPath=1; Kuka.CurrentCDSetIndex=0; Kuka.MovementParameterFieldEnabled=True; IlfCommand=LIN
;ENDFOLD
$BWDSTART = FALSE
LDAT_ACT=LCPDATP88
FDAT_ACT=FP88
BAS (#CP_PARAMS,1)
SET_CD_PARAMS (0)
LIN XP88 C_DIS

;ENDFOLD
;FOLD CIRC CAux89 CDes89 CONT Vel=0.1 m/s CPDATC89 Tool[2] Base[10] ;%{PE}
;FOLD Parameters ;%{h}
;Params IlfProvider=kukaroboter.basistech.inlineforms.movement.old; Kuka.IsGlobalPoint=False; Kuka.PointName=CDes89; Kuka.BlendingEnabled=TRUE; Kuka.MoveDataName=CPDATC89; Kuka.VelocityPath=0.1; Kuka.CurrentCDSetIndex=0; Kuka.MovementParameterFieldEnabled=True; IlfCommand=LIN
;ENDFOLD
$BWDSTART = FALSE
LDAT_ACT=LCPDATC89
FDAT_ACT=FC89
$ORI_TYPE = #VAR
$CIRC_TYPE = #PATH
BAS (#CP_PARAMS,0.1)
SET_CD_PARAMS (0)
CIRC XCAux89, XCDes89 C_DIS

;ENDFOLD
;FOLD LIN P90 CONT Vel=1 m/s CPDATP90 Tool[2] Base[10] ;%{PE}
;FOLD Parameters ;%{h}
;Params IlfProvider=kukaroboter.basistech.inlineforms.movement.old; Kuka.IsGlobalPoint=False; Kuka.PointName=P90; Kuka.BlendingEnabled=TRUE; Kuka.MoveDataName=CPDATP90; Kuka.VelocityPath=1; Kuka.CurrentCDSetIndex=0; Kuka.MovementParameterFieldEnabled=True; IlfCommand=LIN
;ENDFOLD
$BWDSTART = FALSE
LDAT_ACT=LCPDATP90
FDAT_ACT=FP90
BAS (#CP_PARAMS,1)
SET_CD_PARAMS (0)
LIN XP90 C_DIS

;ENDFOLD
;FOLD LIN P91 CONT Vel=1 m/s CPDATP91 Tool[2] Base[10] ;%{PE}
;FOLD Parameters ;%{h}
;Params IlfProvider=kukaroboter.basistech.inlineforms.movement.old; Kuka.IsGlobalPoint=False; Kuka.PointName=P91; Kuka.BlendingEnabled=TRUE; Kuka.MoveDataName=CPDATP91; Kuka.VelocityPath=1; Kuka.CurrentCDSetIndex=0; Kuka.MovementParameterFieldEnabled=True; IlfCommand=LIN
;ENDFOLD
$BWDSTART = FALSE
LDAT_ACT=LCPDATP91
FDAT_ACT=FP91
BAS (#CP_PARAMS,1)
SET_CD_PARAMS (0)
LIN XP91 C_DIS

;ENDFOLD
;FOLD CIRC CAux92 CDes92 CONT Vel=0.1 m/s CPDATC92 Tool[2] Base[10] ;%{PE}
;FOLD Parameters ;%{h}
;Params IlfProvider=kukaroboter.basistech.inlineforms.movement.old; Kuka.IsGlobalPoint=False; Kuka.PointName=CDes92; Kuka.BlendingEnabled=TRUE; Kuka.MoveDataName=CPDATC92; Kuka.VelocityPath=0.1; Kuka.CurrentCDSetIndex=0; Kuka.MovementParameterFieldEnabled=True; IlfCommand=LIN
;ENDFOLD
$BWDSTART = FALSE
LDAT_ACT=LCPDATC92
FDAT_ACT=FC92
$ORI_TYPE = #VAR
$CIRC_TYPE = #PATH
BAS (#CP_PARAMS,0.1)
SET_CD_PARAMS (0)
CIRC XCAux92, XCDes92 C_DIS

;ENDFOLD
;FOLD LIN P93 CONT Vel=1 m/s CPDATP93 Tool[2] Base[10] ;%{PE}
;FOLD Parameters ;%{h}
;Params IlfProvider=kukaroboter.basistech.inlineforms.movement.old; Kuka.IsGlobalPoint=False; Kuka.PointName=P93; Kuka.BlendingEnabled=TRUE; Kuka.MoveDataName=CPDATP93; Kuka.VelocityPath=1; Kuka.CurrentCDSetIndex=0; Kuka.MovementParameterFieldEnabled=True; IlfCommand=LIN
;ENDFOLD
$BWDSTART = FALSE
LDAT_ACT=LCPDATP93
FDAT_ACT=FP93
BAS (#CP_PARAMS,1)
SET_CD_PARAMS (0)
LIN XP93 C_DIS

;ENDFOLD
;FOLD LIN P94 CONT Vel=1 m/s CPDATP94 Tool[2] Base[10] ;%{PE}
;FOLD Parameters ;%{h}
;Params IlfProvider=kukaroboter.basistech.inlineforms.movement.old; Kuka.IsGlobalPoint=False; Kuka.PointName=P94; Kuka.BlendingEnabled=TRUE; Kuka.MoveDataName=CPDATP94; Kuka.VelocityPath=1; Kuka.CurrentCDSetIndex=0; Kuka.MovementParameterFieldEnabled=True; IlfCommand=LIN
;ENDFOLD
$BWDSTART = FALSE
LDAT_ACT=LCPDATP94
FDAT_ACT=FP94
BAS (#CP_PARAMS,1)
SET_CD_PARAMS (0)
LIN XP94 C_DIS

;ENDFOLD
;FOLD CIRC CAux95 CDes95 CONT Vel=0.1 m/s CPDATC95 Tool[2] Base[10] ;%{PE}
;FOLD Parameters ;%{h}
;Params IlfProvider=kukaroboter.basistech.inlineforms.movement.old; Kuka.IsGlobalPoint=False; Kuka.PointName=CDes95; Kuka.BlendingEnabled=TRUE; Kuka.MoveDataName=CPDATC95; Kuka.VelocityPath=0.1; Kuka.CurrentCDSetIndex=0; Kuka.MovementParameterFieldEnabled=True; IlfCommand=LIN
;ENDFOLD
$BWDSTART = FALSE
LDAT_ACT=LCPDATC95
FDAT_ACT=FC95
$ORI_TYPE = #VAR
$CIRC_TYPE = #PATH
BAS (#CP_PARAMS,0.1)
SET_CD_PARAMS (0)
CIRC XCAux95, XCDes95 C_DIS

;ENDFOLD
;FOLD LIN P96 CONT Vel=1 m/s CPDATP96 Tool[2] Base[10] ;%{PE}
;FOLD Parameters ;%{h}
;Params IlfProvider=kukaroboter.basistech.inlineforms.movement.old; Kuka.IsGlobalPoint=False; Kuka.PointName=P96; Kuka.BlendingEnabled=TRUE; Kuka.MoveDataName=CPDATP96; Kuka.VelocityPath=1; Kuka.CurrentCDSetIndex=0; Kuka.MovementParameterFieldEnabled=True; IlfCommand=LIN
;ENDFOLD
$BWDSTART = FALSE
LDAT_ACT=LCPDATP96
FDAT_ACT=FP96
BAS (#CP_PARAMS,1)
SET_CD_PARAMS (0)
LIN XP96 C_DIS

;ENDFOLD
;FOLD LIN P97 CONT Vel=1 m/s CPDATP97 Tool[2] Base[10] ;%{PE}
;FOLD Parameters ;%{h}
;Params IlfProvider=kukaroboter.basistech.inlineforms.movement.old; Kuka.IsGlobalPoint=False; Kuka.PointName=P97; Kuka.BlendingEnabled=TRUE; Kuka.MoveDataName=CPDATP97; Kuka.VelocityPath=1; Kuka.CurrentCDSetIndex=0; Kuka.MovementParameterFieldEnabled=True; IlfCommand=LIN
;ENDFOLD
$BWDSTART = FALSE
LDAT_ACT=LCPDATP97
FDAT_ACT=FP97
BAS (#CP_PARAMS,1)
SET_CD_PARAMS (0)
LIN XP97 C_DIS

;ENDFOLD
;FOLD CIRC CAux98 CDes98 CONT Vel=0.1 m/s CPDATC98 Tool[2] Base[10] ;%{PE}
;FOLD Parameters ;%{h}
;Params IlfProvider=kukaroboter.basistech.inlineforms.movement.old; Kuka.IsGlobalPoint=False; Kuka.PointName=CDes98; Kuka.BlendingEnabled=TRUE; Kuka.MoveDataName=CPDATC98; Kuka.VelocityPath=0.1; Kuka.CurrentCDSetIndex=0; Kuka.MovementParameterFieldEnabled=True; IlfCommand=LIN
;ENDFOLD
$BWDSTART = FALSE
LDAT_ACT=LCPDATC98
FDAT_ACT=FC98
$ORI_TYPE = #VAR
$CIRC_TYPE = #PATH
BAS (#CP_PARAMS,0.1)
SET_CD_PARAMS (0)
CIRC XCAux98, XCDes98 C_DIS

;ENDFOLD
;FOLD LIN P99 CONT Vel=1 m/s CPDATP99 Tool[2] Base[10] ;%{PE}
;FOLD Parameters ;%{h}
;Params IlfProvider=kukaroboter.basistech.inlineforms.movement.old; Kuka.IsGlobalPoint=False; Kuka.PointName=P99; Kuka.BlendingEnabled=TRUE; Kuka.MoveDataName=CPDATP99; Kuka.VelocityPath=1; Kuka.CurrentCDSetIndex=0; Kuka.MovementParameterFieldEnabled=True; IlfCommand=LIN
;ENDFOLD
$BWDSTART = FALSE
LDAT_ACT=LCPDATP99
FDAT_ACT=FP99
BAS (#CP_PARAMS,1)
SET_CD_PARAMS (0)
LIN XP99 C_DIS

;ENDFOLD
;FOLD LIN P100 CONT Vel=1 m/s CPDATP100 Tool[2] Base[10] ;%{PE}
;FOLD Parameters ;%{h}
;Params IlfProvider=kukaroboter.basistech.inlineforms.movement.old; Kuka.IsGlobalPoint=False; Kuka.PointName=P100; Kuka.BlendingEnabled=TRUE; Kuka.MoveDataName=CPDATP100; Kuka.VelocityPath=1; Kuka.CurrentCDSetIndex=0; Kuka.MovementParameterFieldEnabled=True; IlfCommand=LIN
;ENDFOLD
$BWDSTART = FALSE
LDAT_ACT=LCPDATP100
FDAT_ACT=FP100
BAS (#CP_PARAMS,1)
SET_CD_PARAMS (0)
LIN XP100 C_DIS

;ENDFOLD
;FOLD CIRC CAux101 CDes101 CONT Vel=0.1 m/s CPDATC101 Tool[2] Base[10] ;%{PE}
;FOLD Parameters ;%{h}
;Params IlfProvider=kukaroboter.basistech.inlineforms.movement.old; Kuka.IsGlobalPoint=False; Kuka.PointName=CDes101; Kuka.BlendingEnabled=TRUE; Kuka.MoveDataName=CPDATC101; Kuka.VelocityPath=0.1; Kuka.CurrentCDSetIndex=0; Kuka.MovementParameterFieldEnabled=True; IlfCommand=LIN
;ENDFOLD
$BWDSTART = FALSE
LDAT_ACT=LCPDATC101
FDAT_ACT=FC101
$ORI_TYPE = #VAR
$CIRC_TYPE = #PATH
BAS (#CP_PARAMS,0.1)
SET_CD_PARAMS (0)
CIRC XCAux101, XCDes101 C_DIS

;ENDFOLD
;FOLD LIN P102 CONT Vel=1 m/s CPDATP102 Tool[2] Base[10] ;%{PE}
;FOLD Parameters ;%{h}
;Params IlfProvider=kukaroboter.basistech.inlineforms.movement.old; Kuka.IsGlobalPoint=False; Kuka.PointName=P102; Kuka.BlendingEnabled=TRUE; Kuka.MoveDataName=CPDATP102; Kuka.VelocityPath=1; Kuka.CurrentCDSetIndex=0; Kuka.MovementParameterFieldEnabled=True; IlfCommand=LIN
;ENDFOLD
$BWDSTART = FALSE
LDAT_ACT=LCPDATP102
FDAT_ACT=FP102
BAS (#CP_PARAMS,1)
SET_CD_PARAMS (0)
LIN XP102 C_DIS

;ENDFOLD
;FOLD LIN P103 CONT Vel=1 m/s CPDATP103 Tool[2] Base[10] ;%{PE}
;FOLD Parameters ;%{h}
;Params IlfProvider=kukaroboter.basistech.inlineforms.movement.old; Kuka.IsGlobalPoint=False; Kuka.PointName=P103; Kuka.BlendingEnabled=TRUE; Kuka.MoveDataName=CPDATP103; Kuka.VelocityPath=1; Kuka.CurrentCDSetIndex=0; Kuka.MovementParameterFieldEnabled=True; IlfCommand=LIN
;ENDFOLD
$BWDSTART = FALSE
LDAT_ACT=LCPDATP103
FDAT_ACT=FP103
BAS (#CP_PARAMS,1)
SET_CD_PARAMS (0)
LIN XP103 C_DIS

;ENDFOLD
;FOLD CIRC CAux104 CDes104 CONT Vel=0.1 m/s CPDATC104 Tool[2] Base[10] ;%{PE}
;FOLD Parameters ;%{h}
;Params IlfProvider=kukaroboter.basistech.inlineforms.movement.old; Kuka.IsGlobalPoint=False; Kuka.PointName=CDes104; Kuka.BlendingEnabled=TRUE; Kuka.MoveDataName=CPDATC104; Kuka.VelocityPath=0.1; Kuka.CurrentCDSetIndex=0; Kuka.MovementParameterFieldEnabled=True; IlfCommand=LIN
;ENDFOLD
$BWDSTART = FALSE
LDAT_ACT=LCPDATC104
FDAT_ACT=FC104
$ORI_TYPE = #VAR
$CIRC_TYPE = #PATH
BAS (#CP_PARAMS,0.1)
SET_CD_PARAMS (0)
CIRC XCAux104, XCDes104 C_DIS

;ENDFOLD
;FOLD LIN P105 CONT Vel=1 m/s CPDATP105 Tool[2] Base[10] ;%{PE}
;FOLD Parameters ;%{h}
;Params IlfProvider=kukaroboter.basistech.inlineforms.movement.old; Kuka.IsGlobalPoint=False; Kuka.PointName=P105; Kuka.BlendingEnabled=TRUE; Kuka.MoveDataName=CPDATP105; Kuka.VelocityPath=1; Kuka.CurrentCDSetIndex=0; Kuka.MovementParameterFieldEnabled=True; IlfCommand=LIN
;ENDFOLD
$BWDSTART = FALSE
LDAT_ACT=LCPDATP105
FDAT_ACT=FP105
BAS (#CP_PARAMS,1)
SET_CD_PARAMS (0)
LIN XP105 C_DIS

;ENDFOLD
;FOLD LIN P106 CONT Vel=1 m/s CPDATP106 Tool[2] Base[10] ;%{PE}
;FOLD Parameters ;%{h}
;Params IlfProvider=kukaroboter.basistech.inlineforms.movement.old; Kuka.IsGlobalPoint=False; Kuka.PointName=P106; Kuka.BlendingEnabled=TRUE; Kuka.MoveDataName=CPDATP106; Kuka.VelocityPath=1; Kuka.CurrentCDSetIndex=0; Kuka.MovementParameterFieldEnabled=True; IlfCommand=LIN
;ENDFOLD
$BWDSTART = FALSE
LDAT_ACT=LCPDATP106
FDAT_ACT=FP106
BAS (#CP_PARAMS,1)
SET_CD_PARAMS (0)
LIN XP106 C_DIS

;ENDFOLD
;FOLD CIRC CAux107 CDes107 CONT Vel=0.1 m/s CPDATC107 Tool[2] Base[10] ;%{PE}
;FOLD Parameters ;%{h}
;Params IlfProvider=kukaroboter.basistech.inlineforms.movement.old; Kuka.IsGlobalPoint=False; Kuka.PointName=CDes107; Kuka.BlendingEnabled=TRUE; Kuka.MoveDataName=CPDATC107; Kuka.VelocityPath=0.1; Kuka.CurrentCDSetIndex=0; Kuka.MovementParameterFieldEnabled=True; IlfCommand=LIN
;ENDFOLD
$BWDSTART = FALSE
LDAT_ACT=LCPDATC107
FDAT_ACT=FC107
$ORI_TYPE = #VAR
$CIRC_TYPE = #PATH
BAS (#CP_PARAMS,0.1)
SET_CD_PARAMS (0)
CIRC XCAux107, XCDes107 C_DIS

;ENDFOLD
;FOLD LIN P108 CONT Vel=1 m/s CPDATP108 Tool[2] Base[10] ;%{PE}
;FOLD Parameters ;%{h}
;Params IlfProvider=kukaroboter.basistech.inlineforms.movement.old; Kuka.IsGlobalPoint=False; Kuka.PointName=P108; Kuka.BlendingEnabled=TRUE; Kuka.MoveDataName=CPDATP108; Kuka.VelocityPath=1; Kuka.CurrentCDSetIndex=0; Kuka.MovementParameterFieldEnabled=True; IlfCommand=LIN
;ENDFOLD
$BWDSTART = FALSE
LDAT_ACT=LCPDATP108
FDAT_ACT=FP108
BAS (#CP_PARAMS,1)
SET_CD_PARAMS (0)
LIN XP108 C_DIS

;ENDFOLD
;FOLD LIN P109 CONT Vel=1 m/s CPDATP109 Tool[2] Base[10] ;%{PE}
;FOLD Parameters ;%{h}
;Params IlfProvider=kukaroboter.basistech.inlineforms.movement.old; Kuka.IsGlobalPoint=False; Kuka.PointName=P109; Kuka.BlendingEnabled=TRUE; Kuka.MoveDataName=CPDATP109; Kuka.VelocityPath=1; Kuka.CurrentCDSetIndex=0; Kuka.MovementParameterFieldEnabled=True; IlfCommand=LIN
;ENDFOLD
$BWDSTART = FALSE
LDAT_ACT=LCPDATP109
FDAT_ACT=FP109
BAS (#CP_PARAMS,1)
SET_CD_PARAMS (0)
LIN XP109 C_DIS

;ENDFOLD
;FOLD CIRC CAux110 CDes110 CONT Vel=0.1 m/s CPDATC110 Tool[2] Base[10] ;%{PE}
;FOLD Parameters ;%{h}
;Params IlfProvider=kukaroboter.basistech.inlineforms.movement.old; Kuka.IsGlobalPoint=False; Kuka.PointName=CDes110; Kuka.BlendingEnabled=TRUE; Kuka.MoveDataName=CPDATC110; Kuka.VelocityPath=0.1; Kuka.CurrentCDSetIndex=0; Kuka.MovementParameterFieldEnabled=True; IlfCommand=LIN
;ENDFOLD
$BWDSTART = FALSE
LDAT_ACT=LCPDATC110
FDAT_ACT=FC110
$ORI_TYPE = #VAR
$CIRC_TYPE = #PATH
BAS (#CP_PARAMS,0.1)
SET_CD_PARAMS (0)
CIRC XCAux110, XCDes110 C_DIS

;ENDFOLD
;FOLD LIN P111 CONT Vel=1 m/s CPDATP111 Tool[2] Base[10] ;%{PE}
;FOLD Parameters ;%{h}
;Params IlfProvider=kukaroboter.basistech.inlineforms.movement.old; Kuka.IsGlobalPoint=False; Kuka.PointName=P111; Kuka.BlendingEnabled=TRUE; Kuka.MoveDataName=CPDATP111; Kuka.VelocityPath=1; Kuka.CurrentCDSetIndex=0; Kuka.MovementParameterFieldEnabled=True; IlfCommand=LIN
;ENDFOLD
$BWDSTART = FALSE
LDAT_ACT=LCPDATP111
FDAT_ACT=FP111
BAS (#CP_PARAMS,1)
SET_CD_PARAMS (0)
LIN XP111 C_DIS

;ENDFOLD
;FOLD LIN P112 CONT Vel=1 m/s CPDATP112 Tool[2] Base[10] ;%{PE}
;FOLD Parameters ;%{h}
;Params IlfProvider=kukaroboter.basistech.inlineforms.movement.old; Kuka.IsGlobalPoint=False; Kuka.PointName=P112; Kuka.BlendingEnabled=TRUE; Kuka.MoveDataName=CPDATP112; Kuka.VelocityPath=1; Kuka.CurrentCDSetIndex=0; Kuka.MovementParameterFieldEnabled=True; IlfCommand=LIN
;ENDFOLD
$BWDSTART = FALSE
LDAT_ACT=LCPDATP112
FDAT_ACT=FP112
BAS (#CP_PARAMS,1)
SET_CD_PARAMS (0)
LIN XP112 C_DIS

;ENDFOLD
;FOLD CIRC CAux113 CDes113 CONT Vel=0.1 m/s CPDATC113 Tool[2] Base[10] ;%{PE}
;FOLD Parameters ;%{h}
;Params IlfProvider=kukaroboter.basistech.inlineforms.movement.old; Kuka.IsGlobalPoint=False; Kuka.PointName=CDes113; Kuka.BlendingEnabled=TRUE; Kuka.MoveDataName=CPDATC113; Kuka.VelocityPath=0.1; Kuka.CurrentCDSetIndex=0; Kuka.MovementParameterFieldEnabled=True; IlfCommand=LIN
;ENDFOLD
$BWDSTART = FALSE
LDAT_ACT=LCPDATC113
FDAT_ACT=FC113
$ORI_TYPE = #VAR
$CIRC_TYPE = #PATH
BAS (#CP_PARAMS,0.1)
SET_CD_PARAMS (0)
CIRC XCAux113, XCDes113 C_DIS

;ENDFOLD
;FOLD LIN P114 CONT Vel=1 m/s CPDATP114 Tool[2] Base[10] ;%{PE}
;FOLD Parameters ;%{h}
;Params IlfProvider=kukaroboter.basistech.inlineforms.movement.old; Kuka.IsGlobalPoint=False; Kuka.PointName=P114; Kuka.BlendingEnabled=TRUE; Kuka.MoveDataName=CPDATP114; Kuka.VelocityPath=1; Kuka.CurrentCDSetIndex=0; Kuka.MovementParameterFieldEnabled=True; IlfCommand=LIN
;ENDFOLD
$BWDSTART = FALSE
LDAT_ACT=LCPDATP114
FDAT_ACT=FP114
BAS (#CP_PARAMS,1)
SET_CD_PARAMS (0)
LIN XP114 C_DIS

;ENDFOLD
;FOLD LIN P115 CONT Vel=1 m/s CPDATP115 Tool[2] Base[10] ;%{PE}
;FOLD Parameters ;%{h}
;Params IlfProvider=kukaroboter.basistech.inlineforms.movement.old; Kuka.IsGlobalPoint=False; Kuka.PointName=P115; Kuka.BlendingEnabled=TRUE; Kuka.MoveDataName=CPDATP115; Kuka.VelocityPath=1; Kuka.CurrentCDSetIndex=0; Kuka.MovementParameterFieldEnabled=True; IlfCommand=LIN
;ENDFOLD
$BWDSTART = FALSE
LDAT_ACT=LCPDATP115
FDAT_ACT=FP115
BAS (#CP_PARAMS,1)
SET_CD_PARAMS (0)
LIN XP115 C_DIS

;ENDFOLD
;FOLD CIRC CAux116 CDes116 CONT Vel=0.1 m/s CPDATC116 Tool[2] Base[10] ;%{PE}
;FOLD Parameters ;%{h}
;Params IlfProvider=kukaroboter.basistech.inlineforms.movement.old; Kuka.IsGlobalPoint=False; Kuka.PointName=CDes116; Kuka.BlendingEnabled=TRUE; Kuka.MoveDataName=CPDATC116; Kuka.VelocityPath=0.1; Kuka.CurrentCDSetIndex=0; Kuka.MovementParameterFieldEnabled=True; IlfCommand=LIN
;ENDFOLD
$BWDSTART = FALSE
LDAT_ACT=LCPDATC116
FDAT_ACT=FC116
$ORI_TYPE = #VAR
$CIRC_TYPE = #PATH
BAS (#CP_PARAMS,0.1)
SET_CD_PARAMS (0)
CIRC XCAux116, XCDes116 C_DIS

;ENDFOLD
;FOLD LIN P117 CONT Vel=1 m/s CPDATP117 Tool[2] Base[10] ;%{PE}
;FOLD Parameters ;%{h}
;Params IlfProvider=kukaroboter.basistech.inlineforms.movement.old; Kuka.IsGlobalPoint=False; Kuka.PointName=P117; Kuka.BlendingEnabled=TRUE; Kuka.MoveDataName=CPDATP117; Kuka.VelocityPath=1; Kuka.CurrentCDSetIndex=0; Kuka.MovementParameterFieldEnabled=True; IlfCommand=LIN
;ENDFOLD
$BWDSTART = FALSE
LDAT_ACT=LCPDATP117
FDAT_ACT=FP117
BAS (#CP_PARAMS,1)
SET_CD_PARAMS (0)
LIN XP117 C_DIS

;ENDFOLD
;FOLD LIN P118 CONT Vel=1 m/s CPDATP118 Tool[2] Base[10] ;%{PE}
;FOLD Parameters ;%{h}
;Params IlfProvider=kukaroboter.basistech.inlineforms.movement.old; Kuka.IsGlobalPoint=False; Kuka.PointName=P118; Kuka.BlendingEnabled=TRUE; Kuka.MoveDataName=CPDATP118; Kuka.VelocityPath=1; Kuka.CurrentCDSetIndex=0; Kuka.MovementParameterFieldEnabled=True; IlfCommand=LIN
;ENDFOLD
$BWDSTART = FALSE
LDAT_ACT=LCPDATP118
FDAT_ACT=FP118
BAS (#CP_PARAMS,1)
SET_CD_PARAMS (0)
LIN XP118 C_DIS

;ENDFOLD
;FOLD CIRC CAux119 CDes119 CONT Vel=0.1 m/s CPDATC119 Tool[2] Base[10] ;%{PE}
;FOLD Parameters ;%{h}
;Params IlfProvider=kukaroboter.basistech.inlineforms.movement.old; Kuka.IsGlobalPoint=False; Kuka.PointName=CDes119; Kuka.BlendingEnabled=TRUE; Kuka.MoveDataName=CPDATC119; Kuka.VelocityPath=0.1; Kuka.CurrentCDSetIndex=0; Kuka.MovementParameterFieldEnabled=True; IlfCommand=LIN
;ENDFOLD
$BWDSTART = FALSE
LDAT_ACT=LCPDATC119
FDAT_ACT=FC119
$ORI_TYPE = #VAR
$CIRC_TYPE = #PATH
BAS (#CP_PARAMS,0.1)
SET_CD_PARAMS (0)
CIRC XCAux119, XCDes119 C_DIS

;ENDFOLD
;FOLD LIN P120 CONT Vel=1 m/s CPDATP120 Tool[2] Base[10] ;%{PE}
;FOLD Parameters ;%{h}
;Params IlfProvider=kukaroboter.basistech.inlineforms.movement.old; Kuka.IsGlobalPoint=False; Kuka.PointName=P120; Kuka.BlendingEnabled=TRUE; Kuka.MoveDataName=CPDATP120; Kuka.VelocityPath=1; Kuka.CurrentCDSetIndex=0; Kuka.MovementParameterFieldEnabled=True; IlfCommand=LIN
;ENDFOLD
$BWDSTART = FALSE
LDAT_ACT=LCPDATP120
FDAT_ACT=FP120
BAS (#CP_PARAMS,1)
SET_CD_PARAMS (0)
LIN XP120 C_DIS

;ENDFOLD
;FOLD LIN P121 CONT Vel=1 m/s CPDATP121 Tool[2] Base[10] ;%{PE}
;FOLD Parameters ;%{h}
;Params IlfProvider=kukaroboter.basistech.inlineforms.movement.old; Kuka.IsGlobalPoint=False; Kuka.PointName=P121; Kuka.BlendingEnabled=TRUE; Kuka.MoveDataName=CPDATP121; Kuka.VelocityPath=1; Kuka.CurrentCDSetIndex=0; Kuka.MovementParameterFieldEnabled=True; IlfCommand=LIN
;ENDFOLD
$BWDSTART = FALSE
LDAT_ACT=LCPDATP121
FDAT_ACT=FP121
BAS (#CP_PARAMS,1)
SET_CD_PARAMS (0)
LIN XP121 C_DIS

;ENDFOLD
;FOLD CIRC CAux122 CDes122 CONT Vel=0.1 m/s CPDATC122 Tool[2] Base[10] ;%{PE}
;FOLD Parameters ;%{h}
;Params IlfProvider=kukaroboter.basistech.inlineforms.movement.old; Kuka.IsGlobalPoint=False; Kuka.PointName=CDes122; Kuka.BlendingEnabled=TRUE; Kuka.MoveDataName=CPDATC122; Kuka.VelocityPath=0.1; Kuka.CurrentCDSetIndex=0; Kuka.MovementParameterFieldEnabled=True; IlfCommand=LIN
;ENDFOLD
$BWDSTART = FALSE
LDAT_ACT=LCPDATC122
FDAT_ACT=FC122
$ORI_TYPE = #VAR
$CIRC_TYPE = #PATH
BAS (#CP_PARAMS,0.1)
SET_CD_PARAMS (0)
CIRC XCAux122, XCDes122 C_DIS

;ENDFOLD
;FOLD LIN P123 CONT Vel=1 m/s CPDATP123 Tool[2] Base[10] ;%{PE}
;FOLD Parameters ;%{h}
;Params IlfProvider=kukaroboter.basistech.inlineforms.movement.old; Kuka.IsGlobalPoint=False; Kuka.PointName=P123; Kuka.BlendingEnabled=TRUE; Kuka.MoveDataName=CPDATP123; Kuka.VelocityPath=1; Kuka.CurrentCDSetIndex=0; Kuka.MovementParameterFieldEnabled=True; IlfCommand=LIN
;ENDFOLD
$BWDSTART = FALSE
LDAT_ACT=LCPDATP123
FDAT_ACT=FP123
BAS (#CP_PARAMS,1)
SET_CD_PARAMS (0)
LIN XP123 C_DIS

;ENDFOLD
;FOLD LIN P124 CONT Vel=1 m/s CPDATP124 Tool[2] Base[10] ;%{PE}
;FOLD Parameters ;%{h}
;Params IlfProvider=kukaroboter.basistech.inlineforms.movement.old; Kuka.IsGlobalPoint=False; Kuka.PointName=P124; Kuka.BlendingEnabled=TRUE; Kuka.MoveDataName=CPDATP124; Kuka.VelocityPath=1; Kuka.CurrentCDSetIndex=0; Kuka.MovementParameterFieldEnabled=True; IlfCommand=LIN
;ENDFOLD
$BWDSTART = FALSE
LDAT_ACT=LCPDATP124
FDAT_ACT=FP124
BAS (#CP_PARAMS,1)
SET_CD_PARAMS (0)
LIN XP124 C_DIS

;ENDFOLD
;FOLD CIRC CAux125 CDes125 CONT Vel=0.1 m/s CPDATC125 Tool[2] Base[10] ;%{PE}
;FOLD Parameters ;%{h}
;Params IlfProvider=kukaroboter.basistech.inlineforms.movement.old; Kuka.IsGlobalPoint=False; Kuka.PointName=CDes125; Kuka.BlendingEnabled=TRUE; Kuka.MoveDataName=CPDATC125; Kuka.VelocityPath=0.1; Kuka.CurrentCDSetIndex=0; Kuka.MovementParameterFieldEnabled=True; IlfCommand=LIN
;ENDFOLD
$BWDSTART = FALSE
LDAT_ACT=LCPDATC125
FDAT_ACT=FC125
$ORI_TYPE = #VAR
$CIRC_TYPE = #PATH
BAS (#CP_PARAMS,0.1)
SET_CD_PARAMS (0)
CIRC XCAux125, XCDes125 C_DIS

;ENDFOLD
;FOLD LIN P126 CONT Vel=1 m/s CPDATP126 Tool[2] Base[10] ;%{PE}
;FOLD Parameters ;%{h}
;Params IlfProvider=kukaroboter.basistech.inlineforms.movement.old; Kuka.IsGlobalPoint=False; Kuka.PointName=P126; Kuka.BlendingEnabled=TRUE; Kuka.MoveDataName=CPDATP126; Kuka.VelocityPath=1; Kuka.CurrentCDSetIndex=0; Kuka.MovementParameterFieldEnabled=True; IlfCommand=LIN
;ENDFOLD
$BWDSTART = FALSE
LDAT_ACT=LCPDATP126
FDAT_ACT=FP126
BAS (#CP_PARAMS,1)
SET_CD_PARAMS (0)
LIN XP126 C_DIS

;ENDFOLD
;FOLD LIN P127 CONT Vel=1 m/s CPDATP127 Tool[2] Base[10] ;%{PE}
;FOLD Parameters ;%{h}
;Params IlfProvider=kukaroboter.basistech.inlineforms.movement.old; Kuka.IsGlobalPoint=False; Kuka.PointName=P127; Kuka.BlendingEnabled=TRUE; Kuka.MoveDataName=CPDATP127; Kuka.VelocityPath=1; Kuka.CurrentCDSetIndex=0; Kuka.MovementParameterFieldEnabled=True; IlfCommand=LIN
;ENDFOLD
$BWDSTART = FALSE
LDAT_ACT=LCPDATP127
FDAT_ACT=FP127
BAS (#CP_PARAMS,1)
SET_CD_PARAMS (0)
LIN XP127 C_DIS

;ENDFOLD
;FOLD CIRC CAux128 CDes128 CONT Vel=0.1 m/s CPDATC128 Tool[2] Base[10] ;%{PE}
;FOLD Parameters ;%{h}
;Params IlfProvider=kukaroboter.basistech.inlineforms.movement.old; Kuka.IsGlobalPoint=False; Kuka.PointName=CDes128; Kuka.BlendingEnabled=TRUE; Kuka.MoveDataName=CPDATC128; Kuka.VelocityPath=0.1; Kuka.CurrentCDSetIndex=0; Kuka.MovementParameterFieldEnabled=True; IlfCommand=LIN
;ENDFOLD
$BWDSTART = FALSE
LDAT_ACT=LCPDATC128
FDAT_ACT=FC128
$ORI_TYPE = #VAR
$CIRC_TYPE = #PATH
BAS (#CP_PARAMS,0.1)
SET_CD_PARAMS (0)
CIRC XCAux128, XCDes128 C_DIS

;ENDFOLD
;FOLD LIN P129 CONT Vel=1 m/s CPDATP129 Tool[2] Base[10] ;%{PE}
;FOLD Parameters ;%{h}
;Params IlfProvider=kukaroboter.basistech.inlineforms.movement.old; Kuka.IsGlobalPoint=False; Kuka.PointName=P129; Kuka.BlendingEnabled=TRUE; Kuka.MoveDataName=CPDATP129; Kuka.VelocityPath=1; Kuka.CurrentCDSetIndex=0; Kuka.MovementParameterFieldEnabled=True; IlfCommand=LIN
;ENDFOLD
$BWDSTART = FALSE
LDAT_ACT=LCPDATP129
FDAT_ACT=FP129
BAS (#CP_PARAMS,1)
SET_CD_PARAMS (0)
LIN XP129 C_DIS

;ENDFOLD
;FOLD LIN P130 CONT Vel=1 m/s CPDATP130 Tool[2] Base[10] ;%{PE}
;FOLD Parameters ;%{h}
;Params IlfProvider=kukaroboter.basistech.inlineforms.movement.old; Kuka.IsGlobalPoint=False; Kuka.PointName=P130; Kuka.BlendingEnabled=TRUE; Kuka.MoveDataName=CPDATP130; Kuka.VelocityPath=1; Kuka.CurrentCDSetIndex=0; Kuka.MovementParameterFieldEnabled=True; IlfCommand=LIN
;ENDFOLD
$BWDSTART = FALSE
LDAT_ACT=LCPDATP130
FDAT_ACT=FP130
BAS (#CP_PARAMS,1)
SET_CD_PARAMS (0)
LIN XP130 C_DIS

;ENDFOLD
;FOLD CIRC CAux131 CDes131 CONT Vel=0.1 m/s CPDATC131 Tool[2] Base[10] ;%{PE}
;FOLD Parameters ;%{h}
;Params IlfProvider=kukaroboter.basistech.inlineforms.movement.old; Kuka.IsGlobalPoint=False; Kuka.PointName=CDes131; Kuka.BlendingEnabled=TRUE; Kuka.MoveDataName=CPDATC131; Kuka.VelocityPath=0.1; Kuka.CurrentCDSetIndex=0; Kuka.MovementParameterFieldEnabled=True; IlfCommand=LIN
;ENDFOLD
$BWDSTART = FALSE
LDAT_ACT=LCPDATC131
FDAT_ACT=FC131
$ORI_TYPE = #VAR
$CIRC_TYPE = #PATH
BAS (#CP_PARAMS,0.1)
SET_CD_PARAMS (0)
CIRC XCAux131, XCDes131 C_DIS

;ENDFOLD
;FOLD LIN P132 CONT Vel=1 m/s CPDATP132 Tool[2] Base[10] ;%{PE}
;FOLD Parameters ;%{h}
;Params IlfProvider=kukaroboter.basistech.inlineforms.movement.old; Kuka.IsGlobalPoint=False; Kuka.PointName=P132; Kuka.BlendingEnabled=TRUE; Kuka.MoveDataName=CPDATP132; Kuka.VelocityPath=1; Kuka.CurrentCDSetIndex=0; Kuka.MovementParameterFieldEnabled=True; IlfCommand=LIN
;ENDFOLD
$BWDSTART = FALSE
LDAT_ACT=LCPDATP132
FDAT_ACT=FP132
BAS (#CP_PARAMS,1)
SET_CD_PARAMS (0)
LIN XP132 C_DIS

;ENDFOLD
;FOLD LIN P133 CONT Vel=1 m/s CPDATP133 Tool[2] Base[10] ;%{PE}
;FOLD Parameters ;%{h}
;Params IlfProvider=kukaroboter.basistech.inlineforms.movement.old; Kuka.IsGlobalPoint=False; Kuka.PointName=P133; Kuka.BlendingEnabled=TRUE; Kuka.MoveDataName=CPDATP133; Kuka.VelocityPath=1; Kuka.CurrentCDSetIndex=0; Kuka.MovementParameterFieldEnabled=True; IlfCommand=LIN
;ENDFOLD
$BWDSTART = FALSE
LDAT_ACT=LCPDATP133
FDAT_ACT=FP133
BAS (#CP_PARAMS,1)
SET_CD_PARAMS (0)
LIN XP133 C_DIS

;ENDFOLD
;FOLD CIRC CAux134 CDes134 CONT Vel=0.1 m/s CPDATC134 Tool[2] Base[10] ;%{PE}
;FOLD Parameters ;%{h}
;Params IlfProvider=kukaroboter.basistech.inlineforms.movement.old; Kuka.IsGlobalPoint=False; Kuka.PointName=CDes134; Kuka.BlendingEnabled=TRUE; Kuka.MoveDataName=CPDATC134; Kuka.VelocityPath=0.1; Kuka.CurrentCDSetIndex=0; Kuka.MovementParameterFieldEnabled=True; IlfCommand=LIN
;ENDFOLD
$BWDSTART = FALSE
LDAT_ACT=LCPDATC134
FDAT_ACT=FC134
$ORI_TYPE = #VAR
$CIRC_TYPE = #PATH
BAS (#CP_PARAMS,0.1)
SET_CD_PARAMS (0)
CIRC XCAux134, XCDes134 C_DIS

;ENDFOLD
;FOLD LIN P135 CONT Vel=1 m/s CPDATP135 Tool[2] Base[10] ;%{PE}
;FOLD Parameters ;%{h}
;Params IlfProvider=kukaroboter.basistech.inlineforms.movement.old; Kuka.IsGlobalPoint=False; Kuka.PointName=P135; Kuka.BlendingEnabled=TRUE; Kuka.MoveDataName=CPDATP135; Kuka.VelocityPath=1; Kuka.CurrentCDSetIndex=0; Kuka.MovementParameterFieldEnabled=True; IlfCommand=LIN
;ENDFOLD
$BWDSTART = FALSE
LDAT_ACT=LCPDATP135
FDAT_ACT=FP135
BAS (#CP_PARAMS,1)
SET_CD_PARAMS (0)
LIN XP135 C_DIS

;ENDFOLD
;FOLD LIN P136 CONT Vel=1 m/s CPDATP136 Tool[2] Base[10] ;%{PE}
;FOLD Parameters ;%{h}
;Params IlfProvider=kukaroboter.basistech.inlineforms.movement.old; Kuka.IsGlobalPoint=False; Kuka.PointName=P136; Kuka.BlendingEnabled=TRUE; Kuka.MoveDataName=CPDATP136; Kuka.VelocityPath=1; Kuka.CurrentCDSetIndex=0; Kuka.MovementParameterFieldEnabled=True; IlfCommand=LIN
;ENDFOLD
$BWDSTART = FALSE
LDAT_ACT=LCPDATP136
FDAT_ACT=FP136
BAS (#CP_PARAMS,1)
SET_CD_PARAMS (0)
LIN XP136 C_DIS

;ENDFOLD
;FOLD CIRC CAux137 CDes137 CONT Vel=0.1 m/s CPDATC137 Tool[2] Base[10] ;%{PE}
;FOLD Parameters ;%{h}
;Params IlfProvider=kukaroboter.basistech.inlineforms.movement.old; Kuka.IsGlobalPoint=False; Kuka.PointName=CDes137; Kuka.BlendingEnabled=TRUE; Kuka.MoveDataName=CPDATC137; Kuka.VelocityPath=0.1; Kuka.CurrentCDSetIndex=0; Kuka.MovementParameterFieldEnabled=True; IlfCommand=LIN
;ENDFOLD
$BWDSTART = FALSE
LDAT_ACT=LCPDATC137
FDAT_ACT=FC137
$ORI_TYPE = #VAR
$CIRC_TYPE = #PATH
BAS (#CP_PARAMS,0.1)
SET_CD_PARAMS (0)
CIRC XCAux137, XCDes137 C_DIS

;ENDFOLD
;FOLD LIN P138 CONT Vel=1 m/s CPDATP138 Tool[2] Base[10] ;%{PE}
;FOLD Parameters ;%{h}
;Params IlfProvider=kukaroboter.basistech.inlineforms.movement.old; Kuka.IsGlobalPoint=False; Kuka.PointName=P138; Kuka.BlendingEnabled=TRUE; Kuka.MoveDataName=CPDATP138; Kuka.VelocityPath=1; Kuka.CurrentCDSetIndex=0; Kuka.MovementParameterFieldEnabled=True; IlfCommand=LIN
;ENDFOLD
$BWDSTART = FALSE
LDAT_ACT=LCPDATP138
FDAT_ACT=FP138
BAS (#CP_PARAMS,1)
SET_CD_PARAMS (0)
LIN XP138 C_DIS

;ENDFOLD
;FOLD LIN P139 CONT Vel=1 m/s CPDATP139 Tool[2] Base[10] ;%{PE}
;FOLD Parameters ;%{h}
;Params IlfProvider=kukaroboter.basistech.inlineforms.movement.old; Kuka.IsGlobalPoint=False; Kuka.PointName=P139; Kuka.BlendingEnabled=TRUE; Kuka.MoveDataName=CPDATP139; Kuka.VelocityPath=1; Kuka.CurrentCDSetIndex=0; Kuka.MovementParameterFieldEnabled=True; IlfCommand=LIN
;ENDFOLD
$BWDSTART = FALSE
LDAT_ACT=LCPDATP139
FDAT_ACT=FP139
BAS (#CP_PARAMS,1)
SET_CD_PARAMS (0)
LIN XP139 C_DIS

;ENDFOLD
;FOLD CIRC CAux140 CDes140 CONT Vel=0.1 m/s CPDATC140 Tool[2] Base[10] ;%{PE}
;FOLD Parameters ;%{h}
;Params IlfProvider=kukaroboter.basistech.inlineforms.movement.old; Kuka.IsGlobalPoint=False; Kuka.PointName=CDes140; Kuka.BlendingEnabled=TRUE; Kuka.MoveDataName=CPDATC140; Kuka.VelocityPath=0.1; Kuka.CurrentCDSetIndex=0; Kuka.MovementParameterFieldEnabled=True; IlfCommand=LIN
;ENDFOLD
$BWDSTART = FALSE
LDAT_ACT=LCPDATC140
FDAT_ACT=FC140
$ORI_TYPE = #VAR
$CIRC_TYPE = #PATH
BAS (#CP_PARAMS,0.1)
SET_CD_PARAMS (0)
CIRC XCAux140, XCDes140 C_DIS

;ENDFOLD
;FOLD LIN P141 CONT Vel=1 m/s CPDATP141 Tool[2] Base[10] ;%{PE}
;FOLD Parameters ;%{h}
;Params IlfProvider=kukaroboter.basistech.inlineforms.movement.old; Kuka.IsGlobalPoint=False; Kuka.PointName=P141; Kuka.BlendingEnabled=TRUE; Kuka.MoveDataName=CPDATP141; Kuka.VelocityPath=1; Kuka.CurrentCDSetIndex=0; Kuka.MovementParameterFieldEnabled=True; IlfCommand=LIN
;ENDFOLD
$BWDSTART = FALSE
LDAT_ACT=LCPDATP141
FDAT_ACT=FP141
BAS (#CP_PARAMS,1)
SET_CD_PARAMS (0)
LIN XP141 C_DIS

;ENDFOLD
;FOLD LIN P142 CONT Vel=1 m/s CPDATP142 Tool[2] Base[10] ;%{PE}
;FOLD Parameters ;%{h}
;Params IlfProvider=kukaroboter.basistech.inlineforms.movement.old; Kuka.IsGlobalPoint=False; Kuka.PointName=P142; Kuka.BlendingEnabled=TRUE; Kuka.MoveDataName=CPDATP142; Kuka.VelocityPath=1; Kuka.CurrentCDSetIndex=0; Kuka.MovementParameterFieldEnabled=True; IlfCommand=LIN
;ENDFOLD
$BWDSTART = FALSE
LDAT_ACT=LCPDATP142
FDAT_ACT=FP142
BAS (#CP_PARAMS,1)
SET_CD_PARAMS (0)
LIN XP142 C_DIS

;ENDFOLD
;FOLD CIRC CAux143 CDes143 CONT Vel=0.1 m/s CPDATC143 Tool[2] Base[10] ;%{PE}
;FOLD Parameters ;%{h}
;Params IlfProvider=kukaroboter.basistech.inlineforms.movement.old; Kuka.IsGlobalPoint=False; Kuka.PointName=CDes143; Kuka.BlendingEnabled=TRUE; Kuka.MoveDataName=CPDATC143; Kuka.VelocityPath=0.1; Kuka.CurrentCDSetIndex=0; Kuka.MovementParameterFieldEnabled=True; IlfCommand=LIN
;ENDFOLD
$BWDSTART = FALSE
LDAT_ACT=LCPDATC143
FDAT_ACT=FC143
$ORI_TYPE = #VAR
$CIRC_TYPE = #PATH
BAS (#CP_PARAMS,0.1)
SET_CD_PARAMS (0)
CIRC XCAux143, XCDes143 C_DIS

;ENDFOLD
;FOLD LIN P144 CONT Vel=1 m/s CPDATP144 Tool[2] Base[10] ;%{PE}
;FOLD Parameters ;%{h}
;Params IlfProvider=kukaroboter.basistech.inlineforms.movement.old; Kuka.IsGlobalPoint=False; Kuka.PointName=P144; Kuka.BlendingEnabled=TRUE; Kuka.MoveDataName=CPDATP144; Kuka.VelocityPath=1; Kuka.CurrentCDSetIndex=0; Kuka.MovementParameterFieldEnabled=True; IlfCommand=LIN
;ENDFOLD
$BWDSTART = FALSE
LDAT_ACT=LCPDATP144
FDAT_ACT=FP144
BAS (#CP_PARAMS,1)
SET_CD_PARAMS (0)
LIN XP144 C_DIS

;ENDFOLD
;FOLD LIN P145 CONT Vel=1 m/s CPDATP145 Tool[2] Base[10] ;%{PE}
;FOLD Parameters ;%{h}
;Params IlfProvider=kukaroboter.basistech.inlineforms.movement.old; Kuka.IsGlobalPoint=False; Kuka.PointName=P145; Kuka.BlendingEnabled=TRUE; Kuka.MoveDataName=CPDATP145; Kuka.VelocityPath=1; Kuka.CurrentCDSetIndex=0; Kuka.MovementParameterFieldEnabled=True; IlfCommand=LIN
;ENDFOLD
$BWDSTART = FALSE
LDAT_ACT=LCPDATP145
FDAT_ACT=FP145
BAS (#CP_PARAMS,1)
SET_CD_PARAMS (0)
LIN XP145 C_DIS

;ENDFOLD
;FOLD CIRC CAux146 CDes146 CONT Vel=0.1 m/s CPDATC146 Tool[2] Base[10] ;%{PE}
;FOLD Parameters ;%{h}
;Params IlfProvider=kukaroboter.basistech.inlineforms.movement.old; Kuka.IsGlobalPoint=False; Kuka.PointName=CDes146; Kuka.BlendingEnabled=TRUE; Kuka.MoveDataName=CPDATC146; Kuka.VelocityPath=0.1; Kuka.CurrentCDSetIndex=0; Kuka.MovementParameterFieldEnabled=True; IlfCommand=LIN
;ENDFOLD
$BWDSTART = FALSE
LDAT_ACT=LCPDATC146
FDAT_ACT=FC146
$ORI_TYPE = #VAR
$CIRC_TYPE = #PATH
BAS (#CP_PARAMS,0.1)
SET_CD_PARAMS (0)
CIRC XCAux146, XCDes146 C_DIS

;ENDFOLD
;FOLD LIN P147 CONT Vel=1 m/s CPDATP147 Tool[2] Base[10] ;%{PE}
;FOLD Parameters ;%{h}
;Params IlfProvider=kukaroboter.basistech.inlineforms.movement.old; Kuka.IsGlobalPoint=False; Kuka.PointName=P147; Kuka.BlendingEnabled=TRUE; Kuka.MoveDataName=CPDATP147; Kuka.VelocityPath=1; Kuka.CurrentCDSetIndex=0; Kuka.MovementParameterFieldEnabled=True; IlfCommand=LIN
;ENDFOLD
$BWDSTART = FALSE
LDAT_ACT=LCPDATP147
FDAT_ACT=FP147
BAS (#CP_PARAMS,1)
SET_CD_PARAMS (0)
LIN XP147 C_DIS

;ENDFOLD
;FOLD LIN P148 CONT Vel=1 m/s CPDATP148 Tool[2] Base[10] ;%{PE}
;FOLD Parameters ;%{h}
;Params IlfProvider=kukaroboter.basistech.inlineforms.movement.old; Kuka.IsGlobalPoint=False; Kuka.PointName=P148; Kuka.BlendingEnabled=TRUE; Kuka.MoveDataName=CPDATP148; Kuka.VelocityPath=1; Kuka.CurrentCDSetIndex=0; Kuka.MovementParameterFieldEnabled=True; IlfCommand=LIN
;ENDFOLD
$BWDSTART = FALSE
LDAT_ACT=LCPDATP148
FDAT_ACT=FP148
BAS (#CP_PARAMS,1)
SET_CD_PARAMS (0)
LIN XP148 C_DIS

;ENDFOLD
;FOLD CIRC CAux149 CDes149 CONT Vel=0.1 m/s CPDATC149 Tool[2] Base[10] ;%{PE}
;FOLD Parameters ;%{h}
;Params IlfProvider=kukaroboter.basistech.inlineforms.movement.old; Kuka.IsGlobalPoint=False; Kuka.PointName=CDes149; Kuka.BlendingEnabled=TRUE; Kuka.MoveDataName=CPDATC149; Kuka.VelocityPath=0.1; Kuka.CurrentCDSetIndex=0; Kuka.MovementParameterFieldEnabled=True; IlfCommand=LIN
;ENDFOLD
$BWDSTART = FALSE
LDAT_ACT=LCPDATC149
FDAT_ACT=FC149
$ORI_TYPE = #VAR
$CIRC_TYPE = #PATH
BAS (#CP_PARAMS,0.1)
SET_CD_PARAMS (0)
CIRC XCAux149, XCDes149 C_DIS

;ENDFOLD
;FOLD LIN P150 CONT Vel=1 m/s CPDATP150 Tool[2] Base[10] ;%{PE}
;FOLD Parameters ;%{h}
;Params IlfProvider=kukaroboter.basistech.inlineforms.movement.old; Kuka.IsGlobalPoint=False; Kuka.PointName=P150; Kuka.BlendingEnabled=TRUE; Kuka.MoveDataName=CPDATP150; Kuka.VelocityPath=1; Kuka.CurrentCDSetIndex=0; Kuka.MovementParameterFieldEnabled=True; IlfCommand=LIN
;ENDFOLD
$BWDSTART = FALSE
LDAT_ACT=LCPDATP150
FDAT_ACT=FP150
BAS (#CP_PARAMS,1)
SET_CD_PARAMS (0)
LIN XP150 C_DIS

;ENDFOLD
;FOLD LIN P151 CONT Vel=1 m/s CPDATP151 Tool[2] Base[10] ;%{PE}
;FOLD Parameters ;%{h}
;Params IlfProvider=kukaroboter.basistech.inlineforms.movement.old; Kuka.IsGlobalPoint=False; Kuka.PointName=P151; Kuka.BlendingEnabled=TRUE; Kuka.MoveDataName=CPDATP151; Kuka.VelocityPath=1; Kuka.CurrentCDSetIndex=0; Kuka.MovementParameterFieldEnabled=True; IlfCommand=LIN
;ENDFOLD
$BWDSTART = FALSE
LDAT_ACT=LCPDATP151
FDAT_ACT=FP151
BAS (#CP_PARAMS,1)
SET_CD_PARAMS (0)
LIN XP151 C_DIS

;ENDFOLD
;FOLD CIRC CAux152 CDes152 CONT Vel=0.1 m/s CPDATC152 Tool[2] Base[10] ;%{PE}
;FOLD Parameters ;%{h}
;Params IlfProvider=kukaroboter.basistech.inlineforms.movement.old; Kuka.IsGlobalPoint=False; Kuka.PointName=CDes152; Kuka.BlendingEnabled=TRUE; Kuka.MoveDataName=CPDATC152; Kuka.VelocityPath=0.1; Kuka.CurrentCDSetIndex=0; Kuka.MovementParameterFieldEnabled=True; IlfCommand=LIN
;ENDFOLD
$BWDSTART = FALSE
LDAT_ACT=LCPDATC152
FDAT_ACT=FC152
$ORI_TYPE = #VAR
$CIRC_TYPE = #PATH
BAS (#CP_PARAMS,0.1)
SET_CD_PARAMS (0)
CIRC XCAux152, XCDes152 C_DIS

;ENDFOLD
;FOLD LIN P153 CONT Vel=1 m/s CPDATP153 Tool[2] Base[10] ;%{PE}
;FOLD Parameters ;%{h}
;Params IlfProvider=kukaroboter.basistech.inlineforms.movement.old; Kuka.IsGlobalPoint=False; Kuka.PointName=P153; Kuka.BlendingEnabled=TRUE; Kuka.MoveDataName=CPDATP153; Kuka.VelocityPath=1; Kuka.CurrentCDSetIndex=0; Kuka.MovementParameterFieldEnabled=True; IlfCommand=LIN
;ENDFOLD
$BWDSTART = FALSE
LDAT_ACT=LCPDATP153
FDAT_ACT=FP153
BAS (#CP_PARAMS,1)
SET_CD_PARAMS (0)
LIN XP153 C_DIS

;ENDFOLD
;FOLD LIN P154 CONT Vel=1 m/s CPDATP154 Tool[2] Base[10] ;%{PE}
;FOLD Parameters ;%{h}
;Params IlfProvider=kukaroboter.basistech.inlineforms.movement.old; Kuka.IsGlobalPoint=False; Kuka.PointName=P154; Kuka.BlendingEnabled=TRUE; Kuka.MoveDataName=CPDATP154; Kuka.VelocityPath=1; Kuka.CurrentCDSetIndex=0; Kuka.MovementParameterFieldEnabled=True; IlfCommand=LIN
;ENDFOLD
$BWDSTART = FALSE
LDAT_ACT=LCPDATP154
FDAT_ACT=FP154
BAS (#CP_PARAMS,1)
SET_CD_PARAMS (0)
LIN XP154 C_DIS

;ENDFOLD
;FOLD CIRC CAux155 CDes155 CONT Vel=0.1 m/s CPDATC155 Tool[2] Base[10] ;%{PE}
;FOLD Parameters ;%{h}
;Params IlfProvider=kukaroboter.basistech.inlineforms.movement.old; Kuka.IsGlobalPoint=False; Kuka.PointName=CDes155; Kuka.BlendingEnabled=TRUE; Kuka.MoveDataName=CPDATC155; Kuka.VelocityPath=0.1; Kuka.CurrentCDSetIndex=0; Kuka.MovementParameterFieldEnabled=True; IlfCommand=LIN
;ENDFOLD
$BWDSTART = FALSE
LDAT_ACT=LCPDATC155
FDAT_ACT=FC155
$ORI_TYPE = #VAR
$CIRC_TYPE = #PATH
BAS (#CP_PARAMS,0.1)
SET_CD_PARAMS (0)
CIRC XCAux155, XCDes155 C_DIS

;ENDFOLD
;FOLD LIN P156 CONT Vel=1 m/s CPDATP156 Tool[2] Base[10] ;%{PE}
;FOLD Parameters ;%{h}
;Params IlfProvider=kukaroboter.basistech.inlineforms.movement.old; Kuka.IsGlobalPoint=False; Kuka.PointName=P156; Kuka.BlendingEnabled=TRUE; Kuka.MoveDataName=CPDATP156; Kuka.VelocityPath=1; Kuka.CurrentCDSetIndex=0; Kuka.MovementParameterFieldEnabled=True; IlfCommand=LIN
;ENDFOLD
$BWDSTART = FALSE
LDAT_ACT=LCPDATP156
FDAT_ACT=FP156
BAS (#CP_PARAMS,1)
SET_CD_PARAMS (0)
LIN XP156 C_DIS

;ENDFOLD
;FOLD LIN P157 CONT Vel=1 m/s CPDATP157 Tool[2] Base[10] ;%{PE}
;FOLD Parameters ;%{h}
;Params IlfProvider=kukaroboter.basistech.inlineforms.movement.old; Kuka.IsGlobalPoint=False; Kuka.PointName=P157; Kuka.BlendingEnabled=TRUE; Kuka.MoveDataName=CPDATP157; Kuka.VelocityPath=1; Kuka.CurrentCDSetIndex=0; Kuka.MovementParameterFieldEnabled=True; IlfCommand=LIN
;ENDFOLD
$BWDSTART = FALSE
LDAT_ACT=LCPDATP157
FDAT_ACT=FP157
BAS (#CP_PARAMS,1)
SET_CD_PARAMS (0)
LIN XP157 C_DIS

;ENDFOLD
;FOLD CIRC CAux158 CDes158 CONT Vel=0.1 m/s CPDATC158 Tool[2] Base[10] ;%{PE}
;FOLD Parameters ;%{h}
;Params IlfProvider=kukaroboter.basistech.inlineforms.movement.old; Kuka.IsGlobalPoint=False; Kuka.PointName=CDes158; Kuka.BlendingEnabled=TRUE; Kuka.MoveDataName=CPDATC158; Kuka.VelocityPath=0.1; Kuka.CurrentCDSetIndex=0; Kuka.MovementParameterFieldEnabled=True; IlfCommand=LIN
;ENDFOLD
$BWDSTART = FALSE
LDAT_ACT=LCPDATC158
FDAT_ACT=FC158
$ORI_TYPE = #VAR
$CIRC_TYPE = #PATH
BAS (#CP_PARAMS,0.1)
SET_CD_PARAMS (0)
CIRC XCAux158, XCDes158 C_DIS

;ENDFOLD
;FOLD LIN P159 CONT Vel=1 m/s CPDATP159 Tool[2] Base[10] ;%{PE}
;FOLD Parameters ;%{h}
;Params IlfProvider=kukaroboter.basistech.inlineforms.movement.old; Kuka.IsGlobalPoint=False; Kuka.PointName=P159; Kuka.BlendingEnabled=TRUE; Kuka.MoveDataName=CPDATP159; Kuka.VelocityPath=1; Kuka.CurrentCDSetIndex=0; Kuka.MovementParameterFieldEnabled=True; IlfCommand=LIN
;ENDFOLD
$BWDSTART = FALSE
LDAT_ACT=LCPDATP159
FDAT_ACT=FP159
BAS (#CP_PARAMS,1)
SET_CD_PARAMS (0)
LIN XP159 C_DIS

;ENDFOLD
;FOLD LIN P160 CONT Vel=1 m/s CPDATP160 Tool[2] Base[10] ;%{PE}
;FOLD Parameters ;%{h}
;Params IlfProvider=kukaroboter.basistech.inlineforms.movement.old; Kuka.IsGlobalPoint=False; Kuka.PointName=P160; Kuka.BlendingEnabled=TRUE; Kuka.MoveDataName=CPDATP160; Kuka.VelocityPath=1; Kuka.CurrentCDSetIndex=0; Kuka.MovementParameterFieldEnabled=True; IlfCommand=LIN
;ENDFOLD
$BWDSTART = FALSE
LDAT_ACT=LCPDATP160
FDAT_ACT=FP160
BAS (#CP_PARAMS,1)
SET_CD_PARAMS (0)
LIN XP160 C_DIS

;ENDFOLD
;FOLD CIRC CAux161 CDes161 CONT Vel=0.1 m/s CPDATC161 Tool[2] Base[10] ;%{PE}
;FOLD Parameters ;%{h}
;Params IlfProvider=kukaroboter.basistech.inlineforms.movement.old; Kuka.IsGlobalPoint=False; Kuka.PointName=CDes161; Kuka.BlendingEnabled=TRUE; Kuka.MoveDataName=CPDATC161; Kuka.VelocityPath=0.1; Kuka.CurrentCDSetIndex=0; Kuka.MovementParameterFieldEnabled=True; IlfCommand=LIN
;ENDFOLD
$BWDSTART = FALSE
LDAT_ACT=LCPDATC161
FDAT_ACT=FC161
$ORI_TYPE = #VAR
$CIRC_TYPE = #PATH
BAS (#CP_PARAMS,0.1)
SET_CD_PARAMS (0)
CIRC XCAux161, XCDes161 C_DIS

;ENDFOLD
;FOLD LIN P162 CONT Vel=1 m/s CPDATP162 Tool[2] Base[10] ;%{PE}
;FOLD Parameters ;%{h}
;Params IlfProvider=kukaroboter.basistech.inlineforms.movement.old; Kuka.IsGlobalPoint=False; Kuka.PointName=P162; Kuka.BlendingEnabled=TRUE; Kuka.MoveDataName=CPDATP162; Kuka.VelocityPath=1; Kuka.CurrentCDSetIndex=0; Kuka.MovementParameterFieldEnabled=True; IlfCommand=LIN
;ENDFOLD
$BWDSTART = FALSE
LDAT_ACT=LCPDATP162
FDAT_ACT=FP162
BAS (#CP_PARAMS,1)
SET_CD_PARAMS (0)
LIN XP162 C_DIS

;ENDFOLD
;FOLD LIN P163 CONT Vel=1 m/s CPDATP163 Tool[2] Base[10] ;%{PE}
;FOLD Parameters ;%{h}
;Params IlfProvider=kukaroboter.basistech.inlineforms.movement.old; Kuka.IsGlobalPoint=False; Kuka.PointName=P163; Kuka.BlendingEnabled=TRUE; Kuka.MoveDataName=CPDATP163; Kuka.VelocityPath=1; Kuka.CurrentCDSetIndex=0; Kuka.MovementParameterFieldEnabled=True; IlfCommand=LIN
;ENDFOLD
$BWDSTART = FALSE
LDAT_ACT=LCPDATP163
FDAT_ACT=FP163
BAS (#CP_PARAMS,1)
SET_CD_PARAMS (0)
LIN XP163 C_DIS

;ENDFOLD
;FOLD CIRC CAux164 CDes164 CONT Vel=0.1 m/s CPDATC164 Tool[2] Base[10] ;%{PE}
;FOLD Parameters ;%{h}
;Params IlfProvider=kukaroboter.basistech.inlineforms.movement.old; Kuka.IsGlobalPoint=False; Kuka.PointName=CDes164; Kuka.BlendingEnabled=TRUE; Kuka.MoveDataName=CPDATC164; Kuka.VelocityPath=0.1; Kuka.CurrentCDSetIndex=0; Kuka.MovementParameterFieldEnabled=True; IlfCommand=LIN
;ENDFOLD
$BWDSTART = FALSE
LDAT_ACT=LCPDATC164
FDAT_ACT=FC164
$ORI_TYPE = #VAR
$CIRC_TYPE = #PATH
BAS (#CP_PARAMS,0.1)
SET_CD_PARAMS (0)
CIRC XCAux164, XCDes164 C_DIS

;ENDFOLD
;FOLD LIN P165 CONT Vel=1 m/s CPDATP165 Tool[2] Base[10] ;%{PE}
;FOLD Parameters ;%{h}
;Params IlfProvider=kukaroboter.basistech.inlineforms.movement.old; Kuka.IsGlobalPoint=False; Kuka.PointName=P165; Kuka.BlendingEnabled=TRUE; Kuka.MoveDataName=CPDATP165; Kuka.VelocityPath=1; Kuka.CurrentCDSetIndex=0; Kuka.MovementParameterFieldEnabled=True; IlfCommand=LIN
;ENDFOLD
$BWDSTART = FALSE
LDAT_ACT=LCPDATP165
FDAT_ACT=FP165
BAS (#CP_PARAMS,1)
SET_CD_PARAMS (0)
LIN XP165 C_DIS

;ENDFOLD
;FOLD LIN P166 CONT Vel=1 m/s CPDATP166 Tool[2] Base[10] ;%{PE}
;FOLD Parameters ;%{h}
;Params IlfProvider=kukaroboter.basistech.inlineforms.movement.old; Kuka.IsGlobalPoint=False; Kuka.PointName=P166; Kuka.BlendingEnabled=TRUE; Kuka.MoveDataName=CPDATP166; Kuka.VelocityPath=1; Kuka.CurrentCDSetIndex=0; Kuka.MovementParameterFieldEnabled=True; IlfCommand=LIN
;ENDFOLD
$BWDSTART = FALSE
LDAT_ACT=LCPDATP166
FDAT_ACT=FP166
BAS (#CP_PARAMS,1)
SET_CD_PARAMS (0)
LIN XP166 C_DIS

;ENDFOLD
;FOLD CIRC CAux167 CDes167 CONT Vel=0.1 m/s CPDATC167 Tool[2] Base[10] ;%{PE}
;FOLD Parameters ;%{h}
;Params IlfProvider=kukaroboter.basistech.inlineforms.movement.old; Kuka.IsGlobalPoint=False; Kuka.PointName=CDes167; Kuka.BlendingEnabled=TRUE; Kuka.MoveDataName=CPDATC167; Kuka.VelocityPath=0.1; Kuka.CurrentCDSetIndex=0; Kuka.MovementParameterFieldEnabled=True; IlfCommand=LIN
;ENDFOLD
$BWDSTART = FALSE
LDAT_ACT=LCPDATC167
FDAT_ACT=FC167
$ORI_TYPE = #VAR
$CIRC_TYPE = #PATH
BAS (#CP_PARAMS,0.1)
SET_CD_PARAMS (0)
CIRC XCAux167, XCDes167 C_DIS

;ENDFOLD
;FOLD LIN P168 CONT Vel=1 m/s CPDATP168 Tool[2] Base[10] ;%{PE}
;FOLD Parameters ;%{h}
;Params IlfProvider=kukaroboter.basistech.inlineforms.movement.old; Kuka.IsGlobalPoint=False; Kuka.PointName=P168; Kuka.BlendingEnabled=TRUE; Kuka.MoveDataName=CPDATP168; Kuka.VelocityPath=1; Kuka.CurrentCDSetIndex=0; Kuka.MovementParameterFieldEnabled=True; IlfCommand=LIN
;ENDFOLD
$BWDSTART = FALSE
LDAT_ACT=LCPDATP168
FDAT_ACT=FP168
BAS (#CP_PARAMS,1)
SET_CD_PARAMS (0)
LIN XP168 C_DIS

;ENDFOLD
;FOLD LIN P169 CONT Vel=1 m/s CPDATP169 Tool[2] Base[10] ;%{PE}
;FOLD Parameters ;%{h}
;Params IlfProvider=kukaroboter.basistech.inlineforms.movement.old; Kuka.IsGlobalPoint=False; Kuka.PointName=P169; Kuka.BlendingEnabled=TRUE; Kuka.MoveDataName=CPDATP169; Kuka.VelocityPath=1; Kuka.CurrentCDSetIndex=0; Kuka.MovementParameterFieldEnabled=True; IlfCommand=LIN
;ENDFOLD
$BWDSTART = FALSE
LDAT_ACT=LCPDATP169
FDAT_ACT=FP169
BAS (#CP_PARAMS,1)
SET_CD_PARAMS (0)
LIN XP169 C_DIS

;ENDFOLD
;FOLD CIRC CAux170 CDes170 CONT Vel=0.1 m/s CPDATC170 Tool[2] Base[10] ;%{PE}
;FOLD Parameters ;%{h}
;Params IlfProvider=kukaroboter.basistech.inlineforms.movement.old; Kuka.IsGlobalPoint=False; Kuka.PointName=CDes170; Kuka.BlendingEnabled=TRUE; Kuka.MoveDataName=CPDATC170; Kuka.VelocityPath=0.1; Kuka.CurrentCDSetIndex=0; Kuka.MovementParameterFieldEnabled=True; IlfCommand=LIN
;ENDFOLD
$BWDSTART = FALSE
LDAT_ACT=LCPDATC170
FDAT_ACT=FC170
$ORI_TYPE = #VAR
$CIRC_TYPE = #PATH
BAS (#CP_PARAMS,0.1)
SET_CD_PARAMS (0)
CIRC XCAux170, XCDes170 C_DIS

;ENDFOLD
;FOLD LIN P171 CONT Vel=1 m/s CPDATP171 Tool[2] Base[10] ;%{PE}
;FOLD Parameters ;%{h}
;Params IlfProvider=kukaroboter.basistech.inlineforms.movement.old; Kuka.IsGlobalPoint=False; Kuka.PointName=P171; Kuka.BlendingEnabled=TRUE; Kuka.MoveDataName=CPDATP171; Kuka.VelocityPath=1; Kuka.CurrentCDSetIndex=0; Kuka.MovementParameterFieldEnabled=True; IlfCommand=LIN
;ENDFOLD
$BWDSTART = FALSE
LDAT_ACT=LCPDATP171
FDAT_ACT=FP171
BAS (#CP_PARAMS,1)
SET_CD_PARAMS (0)
LIN XP171 C_DIS

;ENDFOLD
;FOLD LIN P172 CONT Vel=1 m/s CPDATP172 Tool[2] Base[10] ;%{PE}
;FOLD Parameters ;%{h}
;Params IlfProvider=kukaroboter.basistech.inlineforms.movement.old; Kuka.IsGlobalPoint=False; Kuka.PointName=P172; Kuka.BlendingEnabled=TRUE; Kuka.MoveDataName=CPDATP172; Kuka.VelocityPath=1; Kuka.CurrentCDSetIndex=0; Kuka.MovementParameterFieldEnabled=True; IlfCommand=LIN
;ENDFOLD
$BWDSTART = FALSE
LDAT_ACT=LCPDATP172
FDAT_ACT=FP172
BAS (#CP_PARAMS,1)
SET_CD_PARAMS (0)
LIN XP172 C_DIS

;ENDFOLD
;FOLD CIRC CAux173 CDes173 CONT Vel=0.1 m/s CPDATC173 Tool[2] Base[10] ;%{PE}
;FOLD Parameters ;%{h}
;Params IlfProvider=kukaroboter.basistech.inlineforms.movement.old; Kuka.IsGlobalPoint=False; Kuka.PointName=CDes173; Kuka.BlendingEnabled=TRUE; Kuka.MoveDataName=CPDATC173; Kuka.VelocityPath=0.1; Kuka.CurrentCDSetIndex=0; Kuka.MovementParameterFieldEnabled=True; IlfCommand=LIN
;ENDFOLD
$BWDSTART = FALSE
LDAT_ACT=LCPDATC173
FDAT_ACT=FC173
$ORI_TYPE = #VAR
$CIRC_TYPE = #PATH
BAS (#CP_PARAMS,0.1)
SET_CD_PARAMS (0)
CIRC XCAux173, XCDes173 C_DIS

;ENDFOLD
;FOLD LIN P174 CONT Vel=1 m/s CPDATP174 Tool[2] Base[10] ;%{PE}
;FOLD Parameters ;%{h}
;Params IlfProvider=kukaroboter.basistech.inlineforms.movement.old; Kuka.IsGlobalPoint=False; Kuka.PointName=P174; Kuka.BlendingEnabled=TRUE; Kuka.MoveDataName=CPDATP174; Kuka.VelocityPath=1; Kuka.CurrentCDSetIndex=0; Kuka.MovementParameterFieldEnabled=True; IlfCommand=LIN
;ENDFOLD
$BWDSTART = FALSE
LDAT_ACT=LCPDATP174
FDAT_ACT=FP174
BAS (#CP_PARAMS,1)
SET_CD_PARAMS (0)
LIN XP174 C_DIS

;ENDFOLD
;FOLD LIN P175 CONT Vel=1 m/s CPDATP175 Tool[2] Base[10] ;%{PE}
;FOLD Parameters ;%{h}
;Params IlfProvider=kukaroboter.basistech.inlineforms.movement.old; Kuka.IsGlobalPoint=False; Kuka.PointName=P175; Kuka.BlendingEnabled=TRUE; Kuka.MoveDataName=CPDATP175; Kuka.VelocityPath=1; Kuka.CurrentCDSetIndex=0; Kuka.MovementParameterFieldEnabled=True; IlfCommand=LIN
;ENDFOLD
$BWDSTART = FALSE
LDAT_ACT=LCPDATP175
FDAT_ACT=FP175
BAS (#CP_PARAMS,1)
SET_CD_PARAMS (0)
LIN XP175 C_DIS

;ENDFOLD
;FOLD CIRC CAux176 CDes176 CONT Vel=0.1 m/s CPDATC176 Tool[2] Base[10] ;%{PE}
;FOLD Parameters ;%{h}
;Params IlfProvider=kukaroboter.basistech.inlineforms.movement.old; Kuka.IsGlobalPoint=False; Kuka.PointName=CDes176; Kuka.BlendingEnabled=TRUE; Kuka.MoveDataName=CPDATC176; Kuka.VelocityPath=0.1; Kuka.CurrentCDSetIndex=0; Kuka.MovementParameterFieldEnabled=True; IlfCommand=LIN
;ENDFOLD
$BWDSTART = FALSE
LDAT_ACT=LCPDATC176
FDAT_ACT=FC176
$ORI_TYPE = #VAR
$CIRC_TYPE = #PATH
BAS (#CP_PARAMS,0.1)
SET_CD_PARAMS (0)
CIRC XCAux176, XCDes176 C_DIS

;ENDFOLD
;FOLD LIN P177 CONT Vel=1 m/s CPDATP177 Tool[2] Base[10] ;%{PE}
;FOLD Parameters ;%{h}
;Params IlfProvider=kukaroboter.basistech.inlineforms.movement.old; Kuka.IsGlobalPoint=False; Kuka.PointName=P177; Kuka.BlendingEnabled=TRUE; Kuka.MoveDataName=CPDATP177; Kuka.VelocityPath=1; Kuka.CurrentCDSetIndex=0; Kuka.MovementParameterFieldEnabled=True; IlfCommand=LIN
;ENDFOLD
$BWDSTART = FALSE
LDAT_ACT=LCPDATP177
FDAT_ACT=FP177
BAS (#CP_PARAMS,1)
SET_CD_PARAMS (0)
LIN XP177 C_DIS

;ENDFOLD
;FOLD LIN P178 CONT Vel=1 m/s CPDATP178 Tool[2] Base[10] ;%{PE}
;FOLD Parameters ;%{h}
;Params IlfProvider=kukaroboter.basistech.inlineforms.movement.old; Kuka.IsGlobalPoint=False; Kuka.PointName=P178; Kuka.BlendingEnabled=TRUE; Kuka.MoveDataName=CPDATP178; Kuka.VelocityPath=1; Kuka.CurrentCDSetIndex=0; Kuka.MovementParameterFieldEnabled=True; IlfCommand=LIN
;ENDFOLD
$BWDSTART = FALSE
LDAT_ACT=LCPDATP178
FDAT_ACT=FP178
BAS (#CP_PARAMS,1)
SET_CD_PARAMS (0)
LIN XP178 C_DIS

;ENDFOLD
;FOLD CIRC CAux179 CDes179 CONT Vel=0.1 m/s CPDATC179 Tool[2] Base[10] ;%{PE}
;FOLD Parameters ;%{h}
;Params IlfProvider=kukaroboter.basistech.inlineforms.movement.old; Kuka.IsGlobalPoint=False; Kuka.PointName=CDes179; Kuka.BlendingEnabled=TRUE; Kuka.MoveDataName=CPDATC179; Kuka.VelocityPath=0.1; Kuka.CurrentCDSetIndex=0; Kuka.MovementParameterFieldEnabled=True; IlfCommand=LIN
;ENDFOLD
$BWDSTART = FALSE
LDAT_ACT=LCPDATC179
FDAT_ACT=FC179
$ORI_TYPE = #VAR
$CIRC_TYPE = #PATH
BAS (#CP_PARAMS,0.1)
SET_CD_PARAMS (0)
CIRC XCAux179, XCDes179 C_DIS

;ENDFOLD
;FOLD LIN P180 CONT Vel=1 m/s CPDATP180 Tool[2] Base[10] ;%{PE}
;FOLD Parameters ;%{h}
;Params IlfProvider=kukaroboter.basistech.inlineforms.movement.old; Kuka.IsGlobalPoint=False; Kuka.PointName=P180; Kuka.BlendingEnabled=TRUE; Kuka.MoveDataName=CPDATP180; Kuka.VelocityPath=1; Kuka.CurrentCDSetIndex=0; Kuka.MovementParameterFieldEnabled=True; IlfCommand=LIN
;ENDFOLD
$BWDSTART = FALSE
LDAT_ACT=LCPDATP180
FDAT_ACT=FP180
BAS (#CP_PARAMS,1)
SET_CD_PARAMS (0)
LIN XP180 C_DIS

;ENDFOLD
;FOLD LIN P181 CONT Vel=1 m/s CPDATP181 Tool[2] Base[10] ;%{PE}
;FOLD Parameters ;%{h}
;Params IlfProvider=kukaroboter.basistech.inlineforms.movement.old; Kuka.IsGlobalPoint=False; Kuka.PointName=P181; Kuka.BlendingEnabled=TRUE; Kuka.MoveDataName=CPDATP181; Kuka.VelocityPath=1; Kuka.CurrentCDSetIndex=0; Kuka.MovementParameterFieldEnabled=True; IlfCommand=LIN
;ENDFOLD
$BWDSTART = FALSE
LDAT_ACT=LCPDATP181
FDAT_ACT=FP181
BAS (#CP_PARAMS,1)
SET_CD_PARAMS (0)
LIN XP181 C_DIS

;ENDFOLD
;FOLD CIRC CAux182 CDes182 CONT Vel=0.1 m/s CPDATC182 Tool[2] Base[10] ;%{PE}
;FOLD Parameters ;%{h}
;Params IlfProvider=kukaroboter.basistech.inlineforms.movement.old; Kuka.IsGlobalPoint=False; Kuka.PointName=CDes182; Kuka.BlendingEnabled=TRUE; Kuka.MoveDataName=CPDATC182; Kuka.VelocityPath=0.1; Kuka.CurrentCDSetIndex=0; Kuka.MovementParameterFieldEnabled=True; IlfCommand=LIN
;ENDFOLD
$BWDSTART = FALSE
LDAT_ACT=LCPDATC182
FDAT_ACT=FC182
$ORI_TYPE = #VAR
$CIRC_TYPE = #PATH
BAS (#CP_PARAMS,0.1)
SET_CD_PARAMS (0)
CIRC XCAux182, XCDes182 C_DIS

;ENDFOLD
;FOLD LIN P183 CONT Vel=1 m/s CPDATP183 Tool[2] Base[10] ;%{PE}
;FOLD Parameters ;%{h}
;Params IlfProvider=kukaroboter.basistech.inlineforms.movement.old; Kuka.IsGlobalPoint=False; Kuka.PointName=P183; Kuka.BlendingEnabled=TRUE; Kuka.MoveDataName=CPDATP183; Kuka.VelocityPath=1; Kuka.CurrentCDSetIndex=0; Kuka.MovementParameterFieldEnabled=True; IlfCommand=LIN
;ENDFOLD
$BWDSTART = FALSE
LDAT_ACT=LCPDATP183
FDAT_ACT=FP183
BAS (#CP_PARAMS,1)
SET_CD_PARAMS (0)
LIN XP183 C_DIS

;ENDFOLD
;FOLD LIN P184 CONT Vel=1 m/s CPDATP184 Tool[2] Base[10] ;%{PE}
;FOLD Parameters ;%{h}
;Params IlfProvider=kukaroboter.basistech.inlineforms.movement.old; Kuka.IsGlobalPoint=False; Kuka.PointName=P184; Kuka.BlendingEnabled=TRUE; Kuka.MoveDataName=CPDATP184; Kuka.VelocityPath=1; Kuka.CurrentCDSetIndex=0; Kuka.MovementParameterFieldEnabled=True; IlfCommand=LIN
;ENDFOLD
$BWDSTART = FALSE
LDAT_ACT=LCPDATP184
FDAT_ACT=FP184
BAS (#CP_PARAMS,1)
SET_CD_PARAMS (0)
LIN XP184 C_DIS

;ENDFOLD
;FOLD CIRC CAux185 CDes185 CONT Vel=0.1 m/s CPDATC185 Tool[2] Base[10] ;%{PE}
;FOLD Parameters ;%{h}
;Params IlfProvider=kukaroboter.basistech.inlineforms.movement.old; Kuka.IsGlobalPoint=False; Kuka.PointName=CDes185; Kuka.BlendingEnabled=TRUE; Kuka.MoveDataName=CPDATC185; Kuka.VelocityPath=0.1; Kuka.CurrentCDSetIndex=0; Kuka.MovementParameterFieldEnabled=True; IlfCommand=LIN
;ENDFOLD
$BWDSTART = FALSE
LDAT_ACT=LCPDATC185
FDAT_ACT=FC185
$ORI_TYPE = #VAR
$CIRC_TYPE = #PATH
BAS (#CP_PARAMS,0.1)
SET_CD_PARAMS (0)
CIRC XCAux185, XCDes185 C_DIS

;ENDFOLD
;FOLD LIN P186 CONT Vel=1 m/s CPDATP186 Tool[2] Base[10] ;%{PE}
;FOLD Parameters ;%{h}
;Params IlfProvider=kukaroboter.basistech.inlineforms.movement.old; Kuka.IsGlobalPoint=False; Kuka.PointName=P186; Kuka.BlendingEnabled=TRUE; Kuka.MoveDataName=CPDATP186; Kuka.VelocityPath=1; Kuka.CurrentCDSetIndex=0; Kuka.MovementParameterFieldEnabled=True; IlfCommand=LIN
;ENDFOLD
$BWDSTART = FALSE
LDAT_ACT=LCPDATP186
FDAT_ACT=FP186
BAS (#CP_PARAMS,1)
SET_CD_PARAMS (0)
LIN XP186 C_DIS

;ENDFOLD
;FOLD LIN P187 CONT Vel=1 m/s CPDATP187 Tool[2] Base[10] ;%{PE}
;FOLD Parameters ;%{h}
;Params IlfProvider=kukaroboter.basistech.inlineforms.movement.old; Kuka.IsGlobalPoint=False; Kuka.PointName=P187; Kuka.BlendingEnabled=TRUE; Kuka.MoveDataName=CPDATP187; Kuka.VelocityPath=1; Kuka.CurrentCDSetIndex=0; Kuka.MovementParameterFieldEnabled=True; IlfCommand=LIN
;ENDFOLD
$BWDSTART = FALSE
LDAT_ACT=LCPDATP187
FDAT_ACT=FP187
BAS (#CP_PARAMS,1)
SET_CD_PARAMS (0)
LIN XP187 C_DIS

;ENDFOLD
;FOLD CIRC CAux188 CDes188 CONT Vel=0.1 m/s CPDATC188 Tool[2] Base[10] ;%{PE}
;FOLD Parameters ;%{h}
;Params IlfProvider=kukaroboter.basistech.inlineforms.movement.old; Kuka.IsGlobalPoint=False; Kuka.PointName=CDes188; Kuka.BlendingEnabled=TRUE; Kuka.MoveDataName=CPDATC188; Kuka.VelocityPath=0.1; Kuka.CurrentCDSetIndex=0; Kuka.MovementParameterFieldEnabled=True; IlfCommand=LIN
;ENDFOLD
$BWDSTART = FALSE
LDAT_ACT=LCPDATC188
FDAT_ACT=FC188
$ORI_TYPE = #VAR
$CIRC_TYPE = #PATH
BAS (#CP_PARAMS,0.1)
SET_CD_PARAMS (0)
CIRC XCAux188, XCDes188 C_DIS

;ENDFOLD
;FOLD LIN P189 CONT Vel=1 m/s CPDATP189 Tool[2] Base[10] ;%{PE}
;FOLD Parameters ;%{h}
;Params IlfProvider=kukaroboter.basistech.inlineforms.movement.old; Kuka.IsGlobalPoint=False; Kuka.PointName=P189; Kuka.BlendingEnabled=TRUE; Kuka.MoveDataName=CPDATP189; Kuka.VelocityPath=1; Kuka.CurrentCDSetIndex=0; Kuka.MovementParameterFieldEnabled=True; IlfCommand=LIN
;ENDFOLD
$BWDSTART = FALSE
LDAT_ACT=LCPDATP189
FDAT_ACT=FP189
BAS (#CP_PARAMS,1)
SET_CD_PARAMS (0)
LIN XP189 C_DIS

;ENDFOLD
;FOLD LIN P190 CONT Vel=1 m/s CPDATP190 Tool[2] Base[10] ;%{PE}
;FOLD Parameters ;%{h}
;Params IlfProvider=kukaroboter.basistech.inlineforms.movement.old; Kuka.IsGlobalPoint=False; Kuka.PointName=P190; Kuka.BlendingEnabled=TRUE; Kuka.MoveDataName=CPDATP190; Kuka.VelocityPath=1; Kuka.CurrentCDSetIndex=0; Kuka.MovementParameterFieldEnabled=True; IlfCommand=LIN
;ENDFOLD
$BWDSTART = FALSE
LDAT_ACT=LCPDATP190
FDAT_ACT=FP190
BAS (#CP_PARAMS,1)
SET_CD_PARAMS (0)
LIN XP190 C_DIS

;ENDFOLD
;FOLD CIRC CAux191 CDes191 CONT Vel=0.1 m/s CPDATC191 Tool[2] Base[10] ;%{PE}
;FOLD Parameters ;%{h}
;Params IlfProvider=kukaroboter.basistech.inlineforms.movement.old; Kuka.IsGlobalPoint=False; Kuka.PointName=CDes191; Kuka.BlendingEnabled=TRUE; Kuka.MoveDataName=CPDATC191; Kuka.VelocityPath=0.1; Kuka.CurrentCDSetIndex=0; Kuka.MovementParameterFieldEnabled=True; IlfCommand=LIN
;ENDFOLD
$BWDSTART = FALSE
LDAT_ACT=LCPDATC191
FDAT_ACT=FC191
$ORI_TYPE = #VAR
$CIRC_TYPE = #PATH
BAS (#CP_PARAMS,0.1)
SET_CD_PARAMS (0)
CIRC XCAux191, XCDes191 C_DIS

;ENDFOLD
;FOLD LIN P192 CONT Vel=1 m/s CPDATP192 Tool[2] Base[10] ;%{PE}
;FOLD Parameters ;%{h}
;Params IlfProvider=kukaroboter.basistech.inlineforms.movement.old; Kuka.IsGlobalPoint=False; Kuka.PointName=P192; Kuka.BlendingEnabled=TRUE; Kuka.MoveDataName=CPDATP192; Kuka.VelocityPath=1; Kuka.CurrentCDSetIndex=0; Kuka.MovementParameterFieldEnabled=True; IlfCommand=LIN
;ENDFOLD
$BWDSTART = FALSE
LDAT_ACT=LCPDATP192
FDAT_ACT=FP192
BAS (#CP_PARAMS,1)
SET_CD_PARAMS (0)
LIN XP192 C_DIS

